  MoveC 1160 to (436.44, -29.66, -5) mm, rotated rx -180 ry 0 rz 5 deg; joints [27.358, -51.401, 157.25, 33.23, -102.458, 8.804] to (420.46, -17.39, -5) mm, rotated rx -180 ry 0 rz 0 deg; joints [25.818, -51.435, 156.847, 26.539, -102.977, 7.092]
  MoveL 1161 to (395.06, -17.39, -5) mm, rotated rx -180 ry 0 rz 0 deg; joints [25.049, -51.607, 155.297, 25.593, -101.516, 6.141]
  MoveL 1162 to (318.86, -17.39, -5) mm, rotated rx -180 ry 0 rz 0 deg; joints [22.982, -51.648, 150.513, 23.174, -97.289, 3.75]
  MoveC 1163 to (306.16, -30.09, -5) mm, rotated rx 180 ry 0 rz 0 deg; joints [21.924, -51.604, 150.031, 22.088, -96.946, 3.432] to (293.46, -17.39, -5) mm, rotated rx -180 ry 0 rz 0 deg; joints [22.363, -51.526, 148.876, 22.483, -95.926, 3.077]
  MoveL 1164 to (191.86, -17.39, -5) mm, rotated rx -180 ry 0 rz 0 deg; joints [20.176, -50.499, 142.119, 20.171, -90.651, 0.831]
  MoveC 1165 to (179.16, -30.09, -5) mm, rotated rx -180 ry 0 rz 0 deg; joints [19.26, -50.373, 141.56, 19.254, -90.251, 0.664] to (166.46, -17.39, -5) mm, rotated rx -180 ry 0 rz 0 deg; joints [19.692, -50.127, 140.379, 19.686, -89.368, 0.357]
  MoveL 1166 to (90.26, -17.39, -5) mm, rotated rx 180 ry 0 rz 0 deg; joints [18.365, -48.779, 135.036, 18.415, -85.578, -0.909]
  MoveL 1167 to (64.86, -17.39, -5) mm, rotated rx -180 ry 0 rz 0 deg; joints [17.96, -48.259, 133.212, 18.045, -84.33, -1.289]
  MoveC 1168 to (61.14, -26.37, -5) mm, rotated rx -180 ry 0 rz 0 deg; joints [17.47, -48.234, 133.149, 17.554, -84.28, -1.26] to (52.16, -30.09, -5) mm, rotated rx 180 ry 0 rz 0 deg; joints [17.156, -48.064, 132.58, 17.251, -83.891, -1.352]
  MoveL 1169 to (52.16, -30.09, -5) mm, rotated rx 180 ry 0 rz 0 deg; joints [17.156, -48.064, 132.58, 17.251, -83.891, -1.352]
  MoveC 1170 to (43.18, -26.37, -5) mm, rotated rx 180 ry 0 rz 0 deg; joints [17.202, -47.846, 131.842, 17.314, -83.396, -1.512] to (39.46, -17.39, -5) mm, rotated rx -180 ry 0 rz 0 deg; joints [17.572, -47.707, 131.366, 17.699, -83.087, -1.652]
  MoveL 1171 to (14.06, -17.39, -5) mm, rotated rx 180 ry 0 rz 0 deg; joints [17.2, -47.124, 129.497, 17.375, -81.847, -1.999]
  MoveC 1172 to (13.61, -17.2, -5) mm, rotated rx -180 ry 0 rz 0 deg; joints [17.202, -47.112, 129.46, 17.378, -81.823, -2.007] to (13.42, -16.75, -5) mm, rotated rx -180 ry 0 rz 0 deg; joints [17.22, -47.105, 129.436, 17.397, -81.807, -2.015]
  MoveL 1173 to (13.42, -16.12, -5) mm, rotated rx 180 ry 0 rz 0 deg; joints [17.25, -47.101, 129.421, 17.428, -81.799, -2.022]
  MoveC 1174 to (13.42, -15.67, -4.81) mm, rotated rx 180 ry 0 rz 0 deg; joints [17.271, -47.111, 129.414, 17.449, -81.782, -2.03] to (13.42, -15.48, -4.37) mm, rotated rx -180 ry 0 rz 0 deg; joints [17.279, -47.143, 129.416, 17.459, -81.755, -2.04]
  Set speed (500.0 mm/s)
  MoveL 1175 to (13.42, -15.48, 5) mm, rotated rx 180 ry 0 rz 0 deg; joints [17.275, -47.829, 129.55, 17.48, -81.228, -2.207]
  MoveL 1176 to (12.15, -16.75, 5) mm, rotated rx -180 ry 0 rz 0 deg; joints [17.198, -47.807, 129.485, 17.404, -81.184, -2.209]
  Set speed (25.4 mm/s)
  MoveL 1177 to (12.15, -16.75, 1) mm, rotated rx 180 ry 0 rz 0 deg; joints [17.2, -47.515, 129.429, 17.395, -81.409, -2.138]
  MoveL 1178 to (12.15, -16.75, -7.72) mm, rotated rx -180 ry 0 rz 0 deg; joints [17.203, -46.876, 129.301, 17.376, -81.897, -1.984]
  MoveC 1179 to (12.34, -16.75, -8.16) mm, rotated rx 180 ry 0 rz 0 deg; joints [17.206, -46.847, 129.308, 17.378, -81.931, -1.974] to (12.79, -16.75, -8.35) mm, rotated rx -180 ry 0 rz 0 deg; joints [17.213, -46.844, 129.338, 17.383, -81.963, -1.964]
  Set speed (50.8 mm/s)
  MoveL 1180 to (13.42, -16.75, -8.35) mm, rotated rx 180 ry 0 rz 0 deg; joints [17.222, -46.859, 129.385, 17.391, -81.994, -1.956]
  MoveC 1181 to (13.87, -16.94, -8.35) mm, rotated rx -180 ry 0 rz 0 deg; joints [17.22, -46.871, 129.423, 17.387, -82.019, -1.948] to (14.06, -17.39, -8.35) mm, rotated rx -180 ry 0 rz 0 deg; joints [17.202, -46.878, 129.447, 17.368, -82.034, -1.941]
  MoveL 1182 to (14.06, -169.79, -8.35) mm, rotated rx 180 ry 0 rz 0 deg; joints [9.897, -47.619, 132.176, 9.952, -83.768, -0.667]
  MoveL 1183 to (471.26, -169.79, -8.35) mm, rotated rx 180 ry 0 rz 30 deg; joints [26.906, -51.035, 156.836, 57.701, -97.685, 13.109]
  MoveL 1184 to (471.26, -17.39, -8.35) mm, rotated rx 180 ry 0 rz 30 deg; joints [35.788, -51.568, 151.463, 65.967, -93.163, 8.832]
  MoveL 1185 to (445.86, -17.39, -8.35) mm, rotated rx -180 ry 0 rz 30 deg; joints [34.843, -51.495, 150.022, 64.967, -92.733, 7.523]
  MoveC 1186 to (436.44, -29.66, -8.35) mm, rotated rx -180 ry 0 rz 5 deg; joints [27.361, -50.987, 157.17, 33.274, -102.738, 8.992] to (420.46, -17.39, -8.35) mm, rotated rx -180 ry 0 rz 0 deg; joints [25.82, -51.025, 156.767, 26.576, -103.273, 7.245]
  MoveL 1187 to (395.06, -17.39, -8.35) mm, rotated rx -180 ry 0 rz 0 deg; joints [25.052, -51.212, 155.221, 25.624, -101.804, 6.282]
  MoveL 1188 to (318.86, -17.39, -8.35) mm, rotated rx -180 ry 0 rz 0 deg; joints [22.985, -51.293, 150.445, 23.19, -97.552, 3.864]
  MoveC 1189 to (306.16, -30.09, -8.35) mm, rotated rx -180 ry 0 rz 0 deg; joints [21.926, -51.253, 149.963, 22.103, -97.208, 3.539] to (293.46, -17.39, -8.35) mm, rotated rx -180 ry 0 rz 0 deg; joints [22.366, -51.184, 148.809, 22.497, -96.181, 3.183]
  MoveL 1190 to (191.86, -17.39, -8.35) mm, rotated rx -180 ry 0 rz 0 deg; joints [20.178, -50.199, 142.06, 20.174, -90.878, 0.914]
  MoveC 1191 to (179.16, -30.09, -8.35) mm, rotated rx -180 ry 0 rz 0 deg; joints [19.262, -50.075, 141.501, 19.256, -90.477, 0.743] to (166.46, -17.39, -8.35) mm, rotated rx -180 ry 0 rz 0 deg; joints [19.693, -49.836, 140.322, 19.687, -89.588, 0.436]
  MoveL 1192 to (90.26, -17.39, -8.35) mm, rotated rx -180 ry 0 rz 0 deg; joints [18.366, -48.512, 134.982, 18.412, -85.781, -0.842]
  MoveL 1193 to (64.86, -17.39, -8.35) mm, rotated rx -180 ry 0 rz 0 deg; joints [17.961, -47.999, 133.16, 18.04, -84.527, -1.225]
  MoveC 1194 to (61.14, -26.37, -8.35) mm, rotated rx 180 ry 0 rz 0 deg; joints [17.472, -47.975, 133.097, 17.549, -84.478, -1.197] to (52.16, -30.09, -8.35) mm, rotated rx 180 ry 0 rz 0 deg; joints [17.158, -47.807, 132.528, 17.246, -84.088, -1.291]
  MoveL 1195 to (52.16, -30.09, -8.35) mm, rotated rx 180 ry 0 rz 0 deg; joints [17.158, -47.807, 132.528, 17.246, -84.088, -1.291]
  MoveC 1196 to (43.18, -26.37, -8.35) mm, rotated rx 180 ry 0 rz 0 deg; joints [17.203, -47.591, 131.79, 17.309, -83.59, -1.451] to (39.46, -17.39, -8.35) mm, rotated rx 180 ry 0 rz 0 deg; joints [17.574, -47.454, 131.315, 17.693, -83.279, -1.591]
  MoveL 1197 to (14.06, -17.39, -8.35) mm, rotated rx -180 ry 0 rz 0 deg; joints [17.202, -46.878, 129.447, 17.368, -82.034, -1.941]
  MoveC 1198 to (13.61, -17.2, -8.35) mm, rotated rx -180 ry 0 rz 0 deg; joints [17.204, -46.866, 129.409, 17.372, -82.009, -1.949] to (13.42, -16.75, -8.35) mm, rotated rx -180 ry 0 rz 0 deg; joints [17.222, -46.859, 129.385, 17.391, -81.994, -1.956]
  MoveL 1199 to (13.42, -16.12, -8.35) mm, rotated rx -180 ry 0 rz 0 deg; joints [17.251, -46.855, 129.371, 17.421, -81.986, -1.963]
  MoveC 1200 to (13.42, -15.67, -8.16) mm, rotated rx -180 ry 0 rz 0 deg; joints [17.272, -46.866, 129.363, 17.442, -81.969, -1.971] to (13.42, -15.48, -7.72) mm, rotated rx 180 ry 0 rz 0 deg; joints [17.28, -46.897, 129.366, 17.452, -81.941, -1.981]
  Set speed (500.0 mm/s)
  MoveL 1201 to (13.42, -15.48, 6) mm, rotated rx 180 ry 0 rz 0 deg; joints [17.274, -47.903, 129.564, 17.482, -81.171, -2.225]
  MoveL 1202 to (-18.41, -15.48, 6) mm, rotated rx -180 ry 0 rz 0 deg; joints [16.828, -47.103, 127.185, 17.109, -79.642, -2.632]
  Set speed (25.4 mm/s)
  MoveL 1203 to (-18.41, -15.48, -4.36) mm, rotated rx 180 ry 0 rz 0 deg; joints [16.832, -46.367, 127.04, 17.083, -80.207, -2.457]
  MoveC 1204 to (-18.41, -15.67, -4.81) mm, rotated rx -180 ry 0 rz 0 deg; joints [16.824, -46.337, 127.038, 17.073, -80.234, -2.447] to (-18.41, -16.12, -5) mm, rotated rx 180 ry 0 rz 0 deg; joints [16.804, -46.327, 127.045, 17.051, -80.249, -2.439]
  Set speed (50.8 mm/s)
  MoveL 1205 to (-18.41, -16.75, -5) mm, rotated rx 180 ry 0 rz 0 deg; joints [16.775, -46.331, 127.06, 17.022, -80.258, -2.431]
  MoveC 1206 to (-18.6, -17.2, -5) mm, rotated rx 180 ry 0 rz 0 deg; joints [16.752, -46.33, 127.056, 16.999, -80.254, -2.428] to (-19.04, -17.39, -5) mm, rotated rx -180 ry 0 rz 0 deg; joints [16.738, -46.32, 127.026, 16.985, -80.235, -2.432]
  MoveL 1207 to (-39.46, -17.39, -5) mm, rotated rx -180 ry 0 rz 0 deg; joints [16.465, -45.799, 125.482, 16.762, -79.242, -2.689]
  MoveC 1208 to (-52.16, -30.09, -5) mm, rotated rx -180 ry 0 rz 0 deg; joints [15.736, -45.554, 124.79, 16.045, -78.775, -2.687] to (-64.86, -17.39, -5) mm, rotated rx -180 ry 0 rz 0 deg; joints [16.136, -45.126, 123.537, 16.501, -78.005, -2.999]
  MoveL 1209 to (-90.26, -17.39, -5) mm, rotated rx 180 ry 0 rz 0 deg; joints [15.821, -44.425, 121.565, 16.258, -76.767, -3.301]
  MoveL 1210 to (-166.46, -17.39, -5) mm, rotated rx -180 ry 0 rz 0 deg; joints [14.942, -42.16, 115.477, 15.633, -73.03, -4.165]
  MoveC 1211 to (-179.16, -30.09, -5) mm, rotated rx -180 ry 0 rz 0 deg; joints [14.289, -41.857, 114.706, 14.99, -72.527, -4.103] to (-191.86, -17.39, -5) mm, rotated rx -180 ry 0 rz 0 deg; joints [14.67, -41.351, 113.385, 15.458, -71.772, -4.444]
  MoveL 1212 to (-293.46, -17.39, -5) mm, rotated rx -180 ry 0 rz 0 deg; joints [13.673, -37.838, 104.651, 14.914, -66.642, -5.544]
  MoveC 1213 to (-306.16, -30.09, -5) mm, rotated rx 180 ry 0 rz 0 deg; joints [13.081, -37.473, 103.782, 14.328, -66.095, -5.435] to (-318.86, -17.39, -5) mm, rotated rx 180 ry 0 rz 0 deg; joints [13.444, -36.887, 102.363, 14.818, -65.326, -5.822]
  MoveL 1214 to (-395.06, -17.39, -5) mm, rotated rx -180 ry 0 rz 0 deg; joints [12.8, -33.84, 95.197, 14.628, -61.268, -6.682]
  MoveL 1215 to (-420.46, -17.39, -5) mm, rotated rx -180 ry 0 rz 0 deg; joints [12.599, -32.754, 92.693, 14.601, -59.871, -6.983]
  MoveC 1216 to (-433.16, -30.09, -5) mm, rotated rx -180 ry 0 rz 0 deg; joints [12.059, -32.314, 91.695, 14.061, -59.263, -6.837] to (-445.86, -17.39, -5) mm, rotated rx -180 ry 0 rz 0 deg; joints [12.404, -31.629, 90.122, 14.593, -58.447, -7.295]
  MoveL 1217 to (-471.26, -17.39, -5) mm, rotated rx -180 ry 0 rz 0 deg; joints [12.214, -30.463, 87.478, 14.606, -56.991, -7.62]
  MoveL 1218 to (-471.26, -169.79, -5) mm, rotated rx -180 ry 0 rz 0 deg; joints [6.956, -31.599, 90.168, 8.208, -57.959, -3.998]
  MoveL 1219 to (-14.06, -169.79, -5) mm, rotated rx -180 ry 0 rz 0 deg; joints [9.66, -47.226, 130.101, 9.748, -82.107, -0.931]
  MoveL 1220 to (-14.06, -17.39, -5) mm, rotated rx -180 ry 0 rz 0 deg; joints [16.806, -46.444, 127.401, 17.042, -80.478, -2.368]
  MoveL 1221 to (-19.04, -17.39, -5) mm, rotated rx -180 ry 0 rz 0 deg; joints [16.738, -46.32, 127.026, 16.985, -80.235, -2.432]
  MoveC 1222 to (-19.49, -17.2, -5) mm, rotated rx -180 ry 0 rz 0 deg; joints [16.74, -46.307, 126.988, 16.989, -80.211, -2.44] to (-19.68, -16.75, -5) mm, rotated rx 180 ry 0 rz 0 deg; joints [16.758, -46.299, 126.964, 17.008, -80.196, -2.447]
  MoveL 1223 to (-19.68, -16.12, -5) mm, rotated rx 180 ry 0 rz 0 deg; joints [16.787, -46.295, 126.95, 17.037, -80.188, -2.455]
  MoveC 1224 to (-19.68, -15.67, -4.81) mm, rotated rx 180 ry 0 rz 0 deg; joints [16.807, -46.305, 126.942, 17.058, -80.172, -2.463] to (-19.68, -15.48, -4.37) mm, rotated rx -180 ry 0 rz 0 deg; joints [16.815, -46.336, 126.945, 17.068, -80.145, -2.473]
  Set speed (500.0 mm/s)
  MoveL 1225 to (-19.68, -15.48, 5) mm, rotated rx -180 ry 0 rz 0 deg; joints [16.811, -46.999, 127.076, 17.092, -79.636, -2.631]
  MoveL 1226 to (-18.41, -15.48, 5) mm, rotated rx 180 ry 0 rz 0 deg; joints [16.828, -47.032, 127.172, 17.106, -79.697, -2.615]
  Set speed (25.4 mm/s)
  MoveL 1227 to (-18.41, -15.48, 1) mm, rotated rx 180 ry 0 rz 0 deg; joints [16.83, -46.748, 127.116, 17.096, -79.916, -2.547]
  MoveL 1228 to (-18.41, -15.48, -7.71) mm, rotated rx 180 ry 0 rz 0 deg; joints [16.834, -46.129, 126.991, 17.075, -80.388, -2.401]
  MoveC 1229 to (-18.41, -15.67, -8.16) mm, rotated rx -180 ry 0 rz 0 deg; joints [16.826, -46.099, 126.989, 17.065, -80.414, -2.391] to (-18.41, -16.12, -8.35) mm, rotated rx -180 ry 0 rz 0 deg; joints [16.805, -46.089, 126.996, 17.043, -80.43, -2.383]
  Set speed (50.8 mm/s)
  MoveL 1230 to (-18.41, -16.75, -8.35) mm, rotated rx -180 ry 0 rz 0 deg; joints [16.777, -46.093, 127.011, 17.014, -80.438, -2.375]
  MoveC 1231 to (-18.6, -17.2, -8.35) mm, rotated rx -180 ry 0 rz 0 deg; joints [16.754, -46.091, 127.007, 16.991, -80.435, -2.373] to (-19.04, -17.39, -8.35) mm, rotated rx 180 ry 0 rz 0 deg; joints [16.739, -46.081, 126.977, 16.977, -80.416, -2.376]
  MoveL 1232 to (-39.46, -17.39, -8.35) mm, rotated rx -180 ry 0 rz 0 deg; joints [16.466, -45.566, 125.433, 16.753, -79.419, -2.635]
  MoveC 1233 to (-52.16, -30.09, -8.35) mm, rotated rx -180 ry 0 rz 0 deg; joints [15.737, -45.323, 124.742, 16.036, -78.951, -2.636] to (-64.86, -17.39, -8.35) mm, rotated rx -180 ry 0 rz 0 deg; joints [16.138, -44.898, 123.489, 16.491, -78.178, -2.947]
  MoveL 1234 to (-90.26, -17.39, -8.35) mm, rotated rx -180 ry 0 rz 0 deg; joints [15.822, -44.203, 121.518, 16.248, -76.935, -3.25]
  MoveL 1235 to (-166.46, -17.39, -8.35) mm, rotated rx 180 ry 0 rz 0 deg; joints [14.943, -41.952, 115.432, 15.621, -73.186, -4.12]
  MoveC 1236 to (-179.16, -30.09, -8.35) mm, rotated rx -180 ry 0 rz 0 deg; joints [14.29, -41.651, 114.66, 14.978, -72.683, -4.059] to (-191.86, -17.39, -8.35) mm, rotated rx -180 ry 0 rz 0 deg; joints [14.671, -41.148, 113.34, 15.445, -71.925, -4.4]
  MoveL 1237 to (-293.46, -17.39, -8.35) mm, rotated rx -180 ry 0 rz 0 deg; joints [13.674, -37.65, 104.607, 14.899, -66.781, -5.504]
  MoveC 1238 to (-306.16, -30.09, -8.35) mm, rotated rx -180 ry 0 rz 0 deg; joints [13.083, -37.286, 103.738, 14.313, -66.233, -5.397] to (-318.86, -17.39, -8.35) mm, rotated rx -180 ry 0 rz 0 deg; joints [13.445, -36.702, 102.319, 14.802, -65.462, -5.783]
  MoveL 1239 to (-395.06, -17.39, -8.35) mm, rotated rx 180 ry 0 rz 0 deg; joints [12.801, -33.665, 95.153, 14.611, -61.395, -6.644]
  MoveL 1240 to (-420.46, -17.39, -8.35) mm, rotated rx -180 ry 0 rz 0 deg; joints [12.6, -32.582, 92.649, 14.583, -59.995, -6.946]
  MoveC 1241 to (-433.16, -30.09, -8.35) mm, rotated rx -180 ry 0 rz 0 deg; joints [12.06, -32.143, 91.65, 14.044, -59.386, -6.802] to (-445.86, -17.39, -8.35) mm, rotated rx -180 ry 0 rz 0 deg; joints [12.405, -31.46, 90.078, 14.575, -58.568, -7.258]
  MoveL 1242 to (-471.26, -17.39, -8.35) mm, rotated rx -180 ry 0 rz 0 deg; joints [12.215, -30.296, 87.433, 14.588, -57.11, -7.583]
  MoveL 1243 to (-471.26, -169.79, -8.35) mm, rotated rx -180 ry 0 rz 0 deg; joints [6.957, -31.429, 90.123, 8.198, -58.082, -3.977]
  MoveL 1244 to (-14.06, -169.79, -8.35) mm, rotated rx 180 ry 0 rz 0 deg; joints [9.661, -46.978, 130.051, 9.745, -82.302, -0.898]
  MoveL 1245 to (-14.06, -17.39, -8.35) mm, rotated rx -180 ry 0 rz 0 deg; joints [16.807, -46.205, 127.352, 17.034, -80.659, -2.312]
  MoveL 1246 to (-19.04, -17.39, -8.35) mm, rotated rx 180 ry 0 rz 0 deg; joints [16.739, -46.081, 126.977, 16.977, -80.416, -2.376]
  MoveC 1247 to (-19.49, -17.2, -8.35) mm, rotated rx -180 ry 0 rz 0 deg; joints [16.741, -46.069, 126.939, 16.981, -80.391, -2.384] to (-19.68, -16.75, -8.35) mm, rotated rx -180 ry 0 rz 0 deg; joints [16.759, -46.061, 126.915, 16.999, -80.376, -2.392]
  MoveL 1248 to (-19.68, -16.12, -8.35) mm, rotated rx -180 ry 0 rz 0 deg; joints [16.788, -46.057, 126.901, 17.029, -80.368, -2.399]
  MoveC 1249 to (-19.68, -15.67, -8.16) mm, rotated rx -180 ry 0 rz 0 deg; joints [16.808, -46.067, 126.893, 17.05, -80.352, -2.407] to (-19.68, -15.48, -7.72) mm, rotated rx -180 ry 0 rz 0 deg; joints [16.816, -46.098, 126.896, 17.06, -80.326, -2.417]
  Set speed (500.0 mm/s)
  MoveL 1250 to (-19.68, -15.48, 6) mm, rotated rx -180 ry 0 rz 0 deg; joints [16.811, -47.07, 127.09, 17.095, -79.581, -2.648]
  MoveL 1251 to (-13.42, -196.52, 6) mm, rotated rx 180 ry 0 rz 0 deg; joints [8.369, -48.146, 130.629, 8.453, -81.694, -0.83]
  Set speed (25.4 mm/s)
  MoveL 1252 to (-13.42, -196.51, -4.36) mm, rotated rx -180 ry 0 rz 0 deg; joints [8.373, -47.375, 130.479, 8.444, -82.309, -0.738]
  MoveC 1253 to (-13.42, -196.7, -4.81) mm, rotated rx -180 ry 0 rz 0 deg; joints [8.364, -47.342, 130.474, 8.435, -82.336, -0.733] to (-13.42, -197.15, -5) mm, rotated rx 180 ry 0 rz 0 deg; joints [8.342, -47.329, 130.477, 8.412, -82.351, -0.728]
  Set speed (50.8 mm/s)
  MoveL 1254 to (-13.42, -197.78, -5) mm, rotated rx -180 ry 0 rz 0 deg; joints [8.311, -47.331, 130.484, 8.381, -82.355, -0.724]
  MoveC 1255 to (-13.61, -198.23, -5) mm, rotated rx -180 ry 0 rz 0 deg; joints [8.288, -47.328, 130.474, 8.358, -82.349, -0.722] to (-14.06, -198.42, -5) mm, rotated rx 180 ry 0 rz 0 deg; joints [8.276, -47.318, 130.442, 8.346, -82.327, -0.723]
  MoveL 1256 to (-39.46, -198.42, -5) mm, rotated rx 180 ry 0 rz 0 deg; joints [8.101, -46.702, 128.494, 8.197, -81.005, -0.894]
  MoveC 1257 to (-52.16, -211.12, -5) mm, rotated rx -180 ry 0 rz 0 deg; joints [7.417, -46.42, 127.644, 7.518, -80.428, -0.872] to (-64.86, -198.42, -5) mm, rotated rx -180 ry 0 rz 0 deg; joints [7.932, -46.056, 126.524, 8.058, -79.691, -1.058]
  MoveL 1258 to (-90.26, -198.42, -5) mm, rotated rx -180 ry 0 rz 0 deg; joints [7.771, -45.379, 124.529, 7.93, -78.381, -1.216]
  MoveL 1259 to (-166.46, -198.42, -5) mm, rotated rx -180 ry 0 rz 0 deg; joints [7.324, -43.178, 118.39, 7.598, -74.466, -1.662]
  MoveC 1260 to (-179.16, -211.12, -5) mm, rotated rx -180 ry 0 rz 0 deg; joints [6.712, -42.83, 117.47, 6.983, -73.878, -1.573] to (-191.86, -198.42, -5) mm, rotated rx -180 ry 0 rz 0 deg; joints [7.186, -42.389, 116.287, 7.505, -73.159, -1.804]
  MoveL 1261 to (-293.46, -198.42, -5) mm, rotated rx -180 ry 0 rz 0 deg; joints [6.683, -38.95, 107.539, 7.211, -67.872, -2.355]
  MoveC 1262 to (-306.16, -211.12, -5) mm, rotated rx -180 ry 0 rz 0 deg; joints [6.128, -38.535, 106.529, 6.642, -67.257, -2.212] to (-318.86, -198.42, -5) mm, rotated rx -180 ry 0 rz 0 deg; joints [6.567, -38.018, 105.256, 7.158, -66.527, -2.491]
  MoveL 1263 to (-395.06, -198.42, -5) mm, rotated rx -180 ry 0 rz 0 deg; joints [6.245, -35.036, 98.132, 7.045, -62.4, -2.909]
  MoveL 1264 to (-420.46, -198.42, -5) mm, rotated rx -180 ry 0 rz 0 deg; joints [6.144, -33.974, 95.651, 7.024, -60.986, -3.054]
  MoveC 1265 to (-433.16, -211.12, -5) mm, rotated rx 180 ry 0 rz 0 deg; joints [5.638, -33.482, 94.518, 6.487, -60.321, -2.864] to (-445.86, -198.42, -5) mm, rotated rx 180 ry 0 rz 0 deg; joints [6.047, -32.876, 93.11, 7.013, -59.549, -3.203]
  MoveL 1266 to (-471.26, -198.42, -5) mm, rotated rx -180 ry 0 rz 0 deg; joints [5.952, -31.738, 90.502, 7.012, -58.084, -3.357]
  MoveL 1267 to (-471.26, -350.82, -5) mm, rotated rx 180 ry 0 rz 0 deg; joints [0.562, -32.088, 91.393, 0.654, -58.436, -0.062]
  MoveL 1268 to (-14.06, -350.82, -5) mm, rotated rx -180 ry 0 rz 0 deg; joints [0.782, -47.534, 131.354, 0.784, -82.952, 0.188]
  MoveL 1269 to (-14.06, -198.42, -5) mm, rotated rx 180 ry 0 rz 0 deg; joints [8.276, -47.318, 130.442, 8.346, -82.327, -0.723]
  MoveC 1270 to (-13.87, -197.97, -5) mm, rotated rx 180 ry 0 rz 0 deg; joints [8.299, -47.321, 130.451, 8.369, -82.333, -0.725] to (-13.42, -197.78, -5) mm, rotated rx -180 ry 0 rz 0 deg; joints [8.311, -47.331, 130.484, 8.381, -82.355, -0.724]
  MoveL 1271 to (-12.79, -197.79, -5) mm, rotated rx 180 ry 0 rz 0 deg; joints [8.316, -47.346, 130.532, 8.385, -82.388, -0.719]
  MoveC 1272 to (-12.34, -197.79, -4.81) mm, rotated rx 180 ry 0 rz 0 deg; joints [8.319, -47.371, 130.569, 8.388, -82.401, -0.718] to (-12.15, -197.78, -4.37) mm, rotated rx -180 ry 0 rz 0 deg; joints [8.32, -47.409, 130.59, 8.39, -82.384, -0.72]
  Set speed (500.0 mm/s)
  MoveL 1273 to (-12.15, -197.79, 5) mm, rotated rx -180 ry 0 rz 0 deg; joints [8.317, -48.107, 130.726, 8.398, -81.828, -0.803]
  MoveL 1274 to (-13.42, -196.51, 5) mm, rotated rx 180 ry 0 rz 0 deg; joints [8.37, -48.072, 130.615, 8.452, -81.754, -0.821]
  Set speed (25.4 mm/s)
  MoveL 1275 to (-13.42, -196.51, 1) mm, rotated rx -180 ry 0 rz 0 deg; joints [8.371, -47.774, 130.558, 8.449, -81.992, -0.785]
  MoveL 1276 to (-13.42, -196.51, -7.71) mm, rotated rx -180 ry 0 rz 0 deg; joints [8.374, -47.125, 130.428, 8.441, -82.505, -0.709]
  MoveC 1277 to (-13.42, -196.7, -8.16) mm, rotated rx -180 ry 0 rz 0 deg; joints [8.365, -47.092, 130.424, 8.432, -82.533, -0.703] to (-13.42, -197.15, -8.35) mm, rotated rx -180 ry 0 rz 0 deg; joints [8.343, -47.08, 130.426, 8.41, -82.547, -0.699]
  Set speed (50.8 mm/s)
  MoveL 1278 to (-13.42, -197.78, -8.35) mm, rotated rx -180 ry 0 rz 0 deg; joints [8.312, -47.082, 130.433, 8.379, -82.552, -0.694]
  MoveC 1279 to (-13.61, -198.23, -8.35) mm, rotated rx 180 ry 0 rz 0 deg; joints [8.289, -47.079, 130.424, 8.355, -82.545, -0.693] to (-14.06, -198.42, -8.35) mm, rotated rx -180 ry 0 rz 0 deg; joints [8.277, -47.069, 130.391, 8.343, -82.523, -0.695]
  MoveL 1280 to (-39.46, -198.42, -8.35) mm, rotated rx -180 ry 0 rz 0 deg; joints [8.102, -46.459, 128.444, 8.194, -81.196, -0.866]
  MoveC 1281 to (-52.16, -211.12, -8.35) mm, rotated rx 180 ry 0 rz 0 deg; joints [7.418, -46.18, 127.595, 7.515, -80.617, -0.846] to (-64.86, -198.42, -8.35) mm, rotated rx -180 ry 0 rz 0 deg; joints [7.934, -45.819, 126.475, 8.055, -79.876, -1.031]
  MoveL 1282 to (-90.26, -198.42, -8.35) mm, rotated rx -180 ry 0 rz 0 deg; joints [7.772, -45.149, 124.481, 7.925, -78.562, -1.19]
  MoveL 1283 to (-166.46, -198.42, -8.35) mm, rotated rx -180 ry 0 rz 0 deg; joints [7.325, -42.964, 118.344, 7.593, -74.633, -1.639]
  MoveC 1284 to (-179.16, -211.12, -8.35) mm, rotated rx 180 ry 0 rz 0 deg; joints [6.713, -42.618, 117.424, 6.978, -74.044, -1.552] to (-191.86, -198.42, -8.35) mm, rotated rx 180 ry 0 rz 0 deg; joints [7.187, -42.179, 116.241, 7.499, -73.321, -1.782]
  MoveL 1285 to (-293.46, -198.42, -8.35) mm, rotated rx 180 ry 0 rz 0 deg; joints [6.683, -38.757, 107.494, 7.205, -68.019, -2.335]
  MoveC 1286 to (-306.16, -211.12, -8.35) mm, rotated rx -180 ry 0 rz 0 deg; joints [6.129, -38.344, 106.485, 6.636, -67.403, -2.194] to (-318.86, -198.42, -8.35) mm, rotated rx -180 ry 0 rz 0 deg; joints [6.568, -37.829, 105.212, 7.151, -66.67, -2.472]
  MoveL 1287 to (-395.06, -198.42, -8.35) mm, rotated rx -180 ry 0 rz 0 deg; joints [6.246, -34.857, 98.088, 7.037, -62.534, -2.891]
  MoveL 1288 to (-420.46, -198.42, -8.35) mm, rotated rx -180 ry 0 rz 0 deg; joints [6.145, -33.798, 95.607, 7.016, -61.117, -3.036]
  MoveC 1289 to (-433.16, -211.12, -8.35) mm, rotated rx -180 ry 0 rz 0 deg; joints [5.639, -33.307, 94.474, 6.48, -60.451, -2.848] to (-445.86, -198.42, -8.35) mm, rotated rx -180 ry 0 rz 0 deg; joints [6.047, -32.703, 93.066, 7.005, -59.676, -3.185]
  MoveL 1290 to (-471.26, -198.42, -8.35) mm, rotated rx -180 ry 0 rz 0 deg; joints [5.953, -31.568, 90.458, 7.003, -58.209, -3.34]
  MoveL 1291 to (-471.26, -350.82, -8.35) mm, rotated rx 180 ry 0 rz 0 deg; joints [0.562, -31.917, 91.348, 0.654, -58.563, -0.06]
  MoveL 1292 to (-14.06, -350.82, -8.35) mm, rotated rx -180 ry 0 rz 0 deg; joints [0.783, -47.281, 131.303, 0.784, -83.153, 0.191]
  MoveL 1293 to (-14.06, -198.42, -8.35) mm, rotated rx -180 ry 0 rz 0 deg; joints [8.277, -47.069, 130.391, 8.343, -82.523, -0.695]
  MoveC 1294 to (-13.87, -197.97, -8.35) mm, rotated rx -180 ry 0 rz 0 deg; joints [8.3, -47.072, 130.401, 8.367, -82.53, -0.696] to (-13.42, -197.78, -8.35) mm, rotated rx -180 ry 0 rz 0 deg; joints [8.312, -47.082, 130.433, 8.379, -82.552, -0.694]
  MoveL 1295 to (-12.79, -197.78, -8.35) mm, rotated rx 180 ry 0 rz 0 deg; joints [8.317, -47.096, 130.481, 8.382, -82.585, -0.69]
  MoveC 1296 to (-12.34, -197.78, -8.16) mm, rotated rx -180 ry 0 rz 0 deg; joints [8.32, -47.121, 130.518, 8.385, -82.598, -0.689] to (-12.15, -197.78, -7.72) mm, rotated rx -180 ry 0 rz 0 deg; joints [8.321, -47.159, 130.539, 8.387, -82.581, -0.691]
  Set speed (500.0 mm/s)
  MoveL 1297 to (-12.15, -197.79, 6) mm, rotated rx -180 ry 0 rz 0 deg; joints [8.317, -48.181, 130.74, 8.399, -81.769, -0.812]
  MoveL 1298 to (12.15, -197.78, 6) mm, rotated rx -180 ry 0 rz 0 deg; joints [8.493, -48.76, 132.585, 8.551, -83.024, -0.644]
  Set speed (25.4 mm/s)
  MoveL 1299 to (12.15, -197.78, -4.36) mm, rotated rx -180 ry 0 rz 0 deg; joints [8.496, -47.967, 132.432, 8.544, -83.656, -0.549]
  MoveC 1300 to (12.34, -197.78, -4.81) mm, rotated rx -180 ry 0 rz 0 deg; joints [8.498, -47.937, 132.439, 8.545, -83.693, -0.543] to (12.79, -197.79, -5) mm, rotated rx 180 ry 0 rz 0 deg; joints [8.501, -47.932, 132.47, 8.548, -83.728, -0.538]
  Set speed (50.8 mm/s)
  MoveL 1301 to (13.42, -197.79, -5) mm, rotated rx 180 ry 0 rz 0 deg; joints [8.506, -47.946, 132.518, 8.552, -83.762, -0.534]
  MoveC 1302 to (13.87, -197.97, -5) mm, rotated rx -180 ry 0 rz 0 deg; joints [8.5, -47.957, 132.554, 8.546, -83.787, -0.529] to (14.06, -198.42, -5) mm, rotated rx 180 ry 0 rz 0 deg; joints [8.479, -47.962, 132.573, 8.524, -83.8, -0.525]
  MoveL 1303 to (14.06, -350.82, -5) mm, rotated rx -180 ry 0 rz 0 deg; joints [0.801, -48.164, 133.496, 0.801, -84.463, 0.207]
  MoveL 1304 to (471.26, -350.82, -5) mm, rotated rx 180 ry 0 rz -60 deg; joints [-17.821, -51.324, 151.408, -77.973, -91.92, -8.972]
  MoveL 1305 to (471.26, -198.42, -5) mm, rotated rx -180 ry 0 rz -60 deg; joints [-7.949, -51.323, 153.756, -68.382, -94.441, -10.657]
  MoveL 1306 to (445.86, -198.42, -5) mm, rotated rx 180 ry 0 rz -60 deg; joints [-7.718, -51.355, 152.031, -68.036, -93.831, -9.004]
  MoveC 1307 to (433.16, -211.12, -5) mm, rotated rx -180 ry 0 rz -60 deg; joints [-8.422, -51.332, 151.038, -68.675, -93.358, -8.147] to (420.46, -198.42, -5) mm, rotated rx -180 ry 0 rz -60 deg; joints [-7.5, -51.304, 150.288, -67.724, -93.229, -7.42]
  MoveL 1308 to (395.06, -198.42, -5) mm, rotated rx -180 ry 0 rz -30 deg; joints [0.228, -50.982, 157.395, -30.724, -103.586, -7.63]
  MoveL 1309 to (318.86, -198.42, -5) mm, rotated rx -180 ry 0 rz 0 deg; joints [11.543, -51.473, 154.194, 11.781, -101.591, 2.85]
  MoveC 1310 to (306.16, -211.12, -5) mm, rotated rx -180 ry 0 rz 0 deg; joints [10.534, -51.491, 153.507, 10.725, -100.942, 2.493] to (293.46, -198.42, -5) mm, rotated rx -180 ry 0 rz 0 deg; joints [11.207, -51.519, 152.489, 11.372, -99.89, 2.423]
  MoveL 1311 to (191.86, -198.42, -5) mm, rotated rx -180 ry 0 rz 0 deg; joints [10.035, -50.954, 145.495, 10.05, -93.602, 1.064]
  MoveC 1312 to (179.16, -211.12, -5) mm, rotated rx 180 ry 0 rz 0 deg; joints [9.17, -50.83, 144.75, 9.178, -93.001, 0.897] to (166.46, -198.42, -5) mm, rotated rx 180 ry 0 rz 0 deg; joints [9.779, -50.661, 143.704, 9.78, -92.129, 0.789]
  MoveL 1313 to (90.26, -198.42, -5) mm, rotated rx 180 ry 0 rz 0 deg; joints [9.083, -49.494, 138.223, 9.084, -87.875, 0.072]
  MoveL 1314 to (64.86, -198.42, -5) mm, rotated rx -180 ry 0 rz 0 deg; joints [8.873, -49.02, 136.359, 8.884, -86.501, -0.139]
  MoveC 1315 to (61.14, -207.4, -5) mm, rotated rx -180 ry 0 rz 0 deg; joints [8.377, -48.969, 136.184, 8.389, -86.375, -0.134] to (52.16, -211.12, -5) mm, rotated rx 180 ry 0 rz 0 deg; joints [8.118, -48.8, 135.558, 8.133, -85.921, -0.186]
  MoveL 1316 to (52.16, -211.12, -5) mm, rotated rx 180 ry 0 rz 0 deg; joints [8.118, -48.8, 135.558, 8.133, -85.921, -0.186]
  MoveC 1317 to (43.18, -207.4, -5) mm, rotated rx 180 ry 0 rz 0 deg; joints [8.242, -48.609, 134.851, 8.264, -85.412, -0.267] to (39.46, -198.42, -5) mm, rotated rx -180 ry 0 rz 0 deg; joints [8.671, -48.509, 134.476, 8.698, -85.143, -0.337]
  MoveL 1318 to (14.06, -198.42, -5) mm, rotated rx -180 ry 0 rz 0 deg; joints [8.479, -47.962, 132.573, 8.524, -83.8, -0.525]
  MoveC 1319 to (13.61, -198.23, -5) mm, rotated rx -180 ry 0 rz 0 deg; joints [8.485, -47.952, 132.537, 8.531, -83.775, -0.53] to (13.42, -197.79, -5) mm, rotated rx 180 ry 0 rz 0 deg; joints [8.506, -47.946, 132.518, 8.552, -83.762, -0.534]
  MoveL 1320 to (13.42, -197.15, -5) mm, rotated rx 180 ry 0 rz 0 deg; joints [8.538, -47.945, 132.511, 8.584, -83.757, -0.538]
  MoveC 1321 to (13.42, -196.7, -4.81) mm, rotated rx 180 ry 0 rz 0 deg; joints [8.56, -47.958, 132.509, 8.606, -83.742, -0.542] to (13.42, -196.52, -4.37) mm, rotated rx -180 ry 0 rz 0 deg; joints [8.569, -47.992, 132.513, 8.616, -83.714, -0.547]
  Set speed (500.0 mm/s)
  MoveL 1322 to (13.42, -196.51, 5) mm, rotated rx -180 ry 0 rz 0 deg; joints [8.566, -48.709, 132.653, 8.623, -83.142, -0.634]
  MoveL 1323 to (12.15, -197.79, 5) mm, rotated rx 180 ry 0 rz 0 deg; joints [8.493, -48.684, 132.571, 8.551, -83.085, -0.635]
  Set speed (25.4 mm/s)
  MoveL 1324 to (12.15, -197.78, 1) mm, rotated rx -180 ry 0 rz 0 deg; joints [8.494, -48.378, 132.513, 8.548, -83.33, -0.598]
  MoveL 1325 to (12.15, -197.78, -7.72) mm, rotated rx -180 ry 0 rz 0 deg; joints [8.498, -47.71, 132.38, 8.542, -83.859, -0.518]
  MoveC 1326 to (12.34, -197.79, -8.16) mm, rotated rx -180 ry 0 rz 0 deg; joints [8.499, -47.68, 132.387, 8.543, -83.896, -0.513] to (12.79, -197.79, -8.35) mm, rotated rx 180 ry 0 rz 0 deg; joints [8.502, -47.675, 132.418, 8.546, -83.931, -0.508]
  Set speed (50.8 mm/s)
  MoveL 1327 to (13.42, -197.79, -8.35) mm, rotated rx -180 ry 0 rz 0 deg; joints [8.507, -47.689, 132.466, 8.55, -83.965, -0.503]
  MoveC 1328 to (13.87, -197.97, -8.35) mm, rotated rx 180 ry 0 rz 0 deg; joints [8.501, -47.7, 132.502, 8.543, -83.99, -0.499] to (14.06, -198.42, -8.35) mm, rotated rx -180 ry 0 rz 0 deg; joints [8.48, -47.705, 132.521, 8.522, -84.003, -0.495]
  MoveL 1329 to (14.06, -350.82, -8.35) mm, rotated rx -180 ry 0 rz 0 deg; joints [0.802, -47.903, 133.444, 0.801, -84.671, 0.21]
  MoveL 1330 to (471.26, -350.82, -8.35) mm, rotated rx 180 ry 0 rz -60 deg; joints [-17.821, -50.962, 151.338, -77.983, -91.981, -9.257]
  MoveL 1331 to (471.26, -198.42, -8.35) mm, rotated rx 180 ry 0 rz -60 deg; joints [-7.948, -50.942, 153.682, -68.404, -94.554, -10.943]
  MoveL 1332 to (445.86, -198.42, -8.35) mm, rotated rx 180 ry 0 rz -60 deg; joints [-7.717, -50.988, 151.959, -68.054, -93.942, -9.278]
  MoveC 1333 to (433.16, -211.12, -8.35) mm, rotated rx -180 ry 0 rz -60 deg; joints [-8.421, -50.973, 150.968, -68.691, -93.463, -8.416] to (420.46, -198.42, -8.35) mm, rotated rx -180 ry 0 rz -60 deg; joints [-7.499, -50.951, 150.219, -67.738, -93.336, -7.683]
  MoveL 1334 to (395.06, -198.42, -8.35) mm, rotated rx -180 ry 0 rz -30 deg; joints [0.23, -50.566, 157.314, -30.764, -103.874, -7.806]
  MoveL 1335 to (318.86, -198.42, -8.35) mm, rotated rx -180 ry 0 rz 0 deg; joints [11.545, -51.088, 154.12, 11.796, -101.895, 2.915]
  MoveC 1336 to (306.16, -211.12, -8.35) mm, rotated rx 180 ry 0 rz 0 deg; joints [10.535, -51.112, 153.433, 10.738, -101.242, 2.551] to (293.46, -198.42, -8.35) mm, rotated rx -180 ry 0 rz 0 deg; joints [11.208, -51.149, 152.418, 11.385, -100.182, 2.483]
  MoveL 1337 to (191.86, -198.42, -8.35) mm, rotated rx -180 ry 0 rz 0 deg; joints [10.036, -50.634, 145.433, 10.054, -93.855, 1.109]
  MoveC 1338 to (179.16, -211.12, -8.35) mm, rotated rx -180 ry 0 rz 0 deg; joints [9.172, -50.515, 144.689, 9.182, -93.251, 0.938] to (166.46, -198.42, -8.35) mm, rotated rx 180 ry 0 rz 0 deg; joints [9.78, -50.352, 143.643, 9.784, -92.374, 0.831]
  MoveL 1339 to (90.26, -198.42, -8.35) mm, rotated rx 180 ry 0 rz 0 deg; joints [9.084, -49.213, 138.167, 9.084, -88.098, 0.107]
  MoveL 1340 to (64.86, -198.42, -8.35) mm, rotated rx -180 ry 0 rz 0 deg; joints [8.874, -48.747, 136.304, 8.883, -86.717, -0.105]
  MoveC 1341 to (61.14, -207.4, -8.35) mm, rotated rx -180 ry 0 rz 0 deg; joints [8.378, -48.697, 136.129, 8.388, -86.59, -0.102] to (52.16, -211.12, -8.35) mm, rotated rx -180 ry 0 rz 0 deg; joints [8.119, -48.531, 135.504, 8.132, -86.134, -0.156]
  MoveL 1342 to (52.16, -211.12, -8.35) mm, rotated rx -180 ry 0 rz 0 deg; joints [8.119, -48.531, 135.504, 8.132, -86.134, -0.156]
  MoveC 1343 to (43.18, -207.4, -8.35) mm, rotated rx -180 ry 0 rz 0 deg; joints [8.243, -48.342, 134.798, 8.263, -85.623, -0.237] to (39.46, -198.42, -8.35) mm, rotated rx -180 ry 0 rz 0 deg; joints [8.673, -48.244, 134.423, 8.696, -85.353, -0.305]
  MoveL 1344 to (14.06, -198.42, -8.35) mm, rotated rx -180 ry 0 rz 0 deg; joints [8.48, -47.705, 132.521, 8.522, -84.003, -0.495]
  MoveC 1345 to (13.61, -198.23, -8.35) mm, rotated rx 180 ry 0 rz 0 deg; joints [8.486, -47.695, 132.485, 8.529, -83.978, -0.499] to (13.42, -197.79, -8.35) mm, rotated rx -180 ry 0 rz 0 deg; joints [8.507, -47.689, 132.466, 8.55, -83.965, -0.503]
  MoveL 1346 to (13.42, -197.15, -8.35) mm, rotated rx -180 ry 0 rz 0 deg; joints [8.539, -47.688, 132.459, 8.582, -83.96, -0.507]
  MoveC 1347 to (13.42, -196.7, -8.16) mm, rotated rx -180 ry 0 rz 0 deg; joints [8.561, -47.701, 132.457, 8.604, -83.945, -0.511] to (13.42, -196.52, -7.72) mm, rotated rx 180 ry 0 rz 0 deg; joints [8.57, -47.735, 132.462, 8.614, -83.916, -0.516]
  Set speed (500.0 mm/s)
  MoveL 1348 to (13.42, -196.52, 6) mm, rotated rx 180 ry 0 rz 0 deg; joints [8.565, -48.786, 132.667, 8.623, -83.08, -0.644]
  MoveL 1349 to (12.15, -384.12, 6) mm, rotated rx -180 ry 0 rz 0 deg; joints [-0.891, -48.964, 133.513, -0.901, -83.68, 0.358]
  Set speed (25.4 mm/s)
  MoveL 1350 to (12.15, -384.12, -4.37) mm, rotated rx -180 ry 0 rz 0 deg; joints [-0.889, -48.159, 133.357, -0.897, -84.329, 0.347]
  MoveC 1351 to (12.34, -384.12, -4.81) mm, rotated rx -180 ry 0 rz 0 deg; joints [-0.889, -48.128, 133.364, -0.897, -84.367, 0.347] to (12.79, -384.12, -5) mm, rotated rx -180 ry 0 rz 0 deg; joints [-0.889, -48.124, 133.395, -0.897, -84.403, 0.346]
  Set speed (50.8 mm/s)
  MoveL 1352 to (13.42, -384.12, -5) mm, rotated rx 180 ry 0 rz 0 deg; joints [-0.89, -48.137, 133.444, -0.898, -84.437, 0.346]
  MoveC 1353 to (13.87, -384.31, -5) mm, rotated rx 180 ry 0 rz 0 deg; joints [-0.899, -48.147, 133.477, -0.908, -84.461, 0.346] to (14.06, -384.76, -5) mm, rotated rx -180 ry 0 rz 0 deg; joints [-0.922, -48.151, 133.491, -0.931, -84.471, 0.348]
  MoveL 1354 to (14.06, -537.16, -5) mm, rotated rx -180 ry 0 rz 0 deg; joints [-8.598, -47.831, 132.519, -8.65, -83.879, 1.07]
  MoveL 1355 to (471.26, -537.16, -5) mm, rotated rx -180 ry 0 rz -30 deg; joints [-25.102, -50.905, 157.482, -56.092, -98.794, -13.027]
  MoveL 1356 to (471.26, -384.76, -5) mm, rotated rx -180 ry 0 rz -60 deg; joints [-19.898, -51.3, 150.649, -80.002, -91.436, -8.316]
  MoveL 1357 to (445.86, -384.76, -5) mm, rotated rx 180 ry 0 rz -60 deg; joints [-19.357, -51.196, 148.981, -79.43, -91.236, -6.763]
  MoveC 1358 to (433.16, -397.46, -5) mm, rotated rx -180 ry 0 rz -60 deg; joints [-19.835, -51.091, 147.842, -79.885, -90.991, -5.756] to (420.46, -384.76, -5) mm, rotated rx -180 ry 0 rz -60 deg; joints [-18.844, -51.03, 147.294, -78.891, -91.011, -5.256]
  MoveL 1359 to (395.06, -384.76, -5) mm, rotated rx 180 ry 0 rz -30 deg; joints [-13.014, -51.124, 155.98, -43.881, -100.196, -9.566]
  MoveL 1360 to (318.86, -384.76, -5) mm, rotated rx -180 ry 0 rz 0 deg; joints [-1.265, -51.255, 155.308, -1.304, -103.18, -0.044]
  MoveC 1361 to (306.16, -397.46, -5) mm, rotated rx -180 ry 0 rz 0 deg; joints [-2.116, -51.32, 154.42, -2.169, -102.221, -0.219] to (293.46, -384.76, -5) mm, rotated rx -180 ry 0 rz 0 deg; joints [-1.227, -51.37, 153.582, -1.256, -101.339, 0.007]
  MoveL 1362 to (191.86, -384.76, -5) mm, rotated rx -180 ry 0 rz 0 deg; joints [-1.096, -50.992, 146.511, -1.103, -94.648, 0.166]
  MoveC 1363 to (179.16, -397.46, -5) mm, rotated rx -180 ry 0 rz 0 deg; joints [-1.836, -50.86, 145.584, -1.844, -93.853, 0.12] to (166.46, -384.76, -5) mm, rotated rx -180 ry 0 rz 0 deg; joints [-1.067, -50.73, 144.702, -1.073, -93.102, 0.198]
  MoveL 1364 to (90.26, -384.76, -5) mm, rotated rx 180 ry 0 rz 0 deg; joints [-0.989, -49.634, 139.177, -0.994, -88.674, 0.28]
  MoveL 1365 to (64.86, -384.76, -5) mm, rotated rx -180 ry 0 rz 0 deg; joints [-0.966, -49.178, 137.3, -0.971, -87.253, 0.304]
  MoveC 1366 to (61.14, -393.74, -5) mm, rotated rx -180 ry 0 rz 0 deg; joints [-1.438, -49.101, 137.009, -1.444, -87.039, 0.325] to (52.16, -397.46, -5) mm, rotated rx -180 ry 0 rz 0 deg; joints [-1.622, -48.925, 136.333, -1.629, -86.539, 0.346]
  MoveL 1367 to (52.16, -397.46, -5) mm, rotated rx -180 ry 0 rz 0 deg; joints [-1.622, -48.925, 136.333, -1.629, -86.539, 0.346]
  MoveC 1368 to (43.18, -393.74, -5) mm, rotated rx 180 ry 0 rz 0 deg; joints [-1.415, -48.751, 135.669, -1.422, -86.049, 0.349] to (39.46, -384.76, -5) mm, rotated rx 180 ry 0 rz 0 deg; joints [-0.944, -48.683, 135.405, -0.95, -85.853, 0.327]
  MoveL 1369 to (14.06, -384.76, -5) mm, rotated rx -180 ry 0 rz 0 deg; joints [-0.922, -48.151, 133.491, -0.931, -84.471, 0.348]
  MoveC 1370 to (13.61, -384.57, -5) mm, rotated rx -180 ry 0 rz 0 deg; joints [-0.913, -48.141, 133.457, -0.921, -84.447, 0.348] to (13.42, -384.12, -5) mm, rotated rx 180 ry 0 rz 0 deg; joints [-0.89, -48.137, 133.444, -0.898, -84.437, 0.346]
  MoveL 1371 to (13.42, -383.49, -5) mm, rotated rx 180 ry 0 rz 0 deg; joints [-0.857, -48.138, 133.444, -0.866, -84.437, 0.343]
  MoveC 1372 to (13.42, -383.04, -4.81) mm, rotated rx -180 ry 0 rz 0 deg; joints [-0.835, -48.153, 133.448, -0.843, -84.426, 0.341] to (13.42, -382.85, -4.37) mm, rotated rx -180 ry 0 rz 0 deg; joints [-0.825, -48.188, 133.455, -0.833, -84.398, 0.341]
  Set speed (500.0 mm/s)
  MoveL 1373 to (13.42, -382.85, 5) mm, rotated rx -180 ry 0 rz 0 deg; joints [-0.827, -48.916, 133.596, -0.836, -83.811, 0.35]
  MoveL 1374 to (12.15, -384.12, 5) mm, rotated rx 180 ry 0 rz 0 deg; joints [-0.891, -48.886, 133.498, -0.9, -83.743, 0.357]
  Set speed (25.4 mm/s)
  MoveL 1375 to (12.15, -384.12, 1) mm, rotated rx -180 ry 0 rz 0 deg; joints [-0.89, -48.576, 133.439, -0.899, -83.994, 0.353]
  MoveL 1376 to (12.15, -384.12, -7.71) mm, rotated rx -180 ry 0 rz 0 deg; joints [-0.888, -47.899, 133.305, -0.896, -84.537, 0.344]
  MoveC 1377 to (12.34, -384.12, -8.16) mm, rotated rx -180 ry 0 rz 0 deg; joints [-0.888, -47.868, 133.312, -0.896, -84.575, 0.344] to (12.79, -384.12, -8.35) mm, rotated rx -180 ry 0 rz 0 deg; joints [-0.888, -47.863, 133.343, -0.896, -84.611, 0.343]
  Set speed (50.8 mm/s)
  MoveL 1378 to (13.42, -384.12, -8.35) mm, rotated rx -180 ry 0 rz 0 deg; joints [-0.889, -47.877, 133.391, -0.897, -84.645, 0.342]
  MoveC 1379 to (13.87, -384.31, -8.35) mm, rotated rx -180 ry 0 rz 0 deg; joints [-0.899, -47.886, 133.425, -0.907, -84.669, 0.343] to (14.06, -384.76, -8.35) mm, rotated rx -180 ry 0 rz 0 deg; joints [-0.922, -47.89, 133.438, -0.93, -84.679, 0.345]
  MoveL 1380 to (14.06, -537.16, -8.35) mm, rotated rx -180 ry 0 rz 0 deg; joints [-8.597, -47.574, 132.467, -8.647, -84.082, 1.039]
  MoveL 1381 to (471.26, -537.16, -8.35) mm, rotated rx -180 ry 0 rz -30 deg; joints [-25.103, -50.488, 157.401, -56.136, -98.981, -13.309]
  MoveL 1382 to (471.26, -384.76, -8.35) mm, rotated rx -180 ry 0 rz -60 deg; joints [-19.899, -50.945, 150.579, -80.009, -91.485, -8.598]
  MoveL 1383 to (445.86, -384.76, -8.35) mm, rotated rx -180 ry 0 rz -60 deg; joints [-19.357, -50.853, 148.914, -79.436, -91.286, -7.034]
  MoveC 1384 to (433.16, -397.46, -8.35) mm, rotated rx -180 ry 0 rz -60 deg; joints [-19.835, -50.756, 147.777, -79.89, -91.038, -6.022] to (420.46, -384.76, -8.35) mm, rotated rx -180 ry 0 rz -60 deg; joints [-18.844, -50.699, 147.229, -78.896, -91.063, -5.518]
  MoveL 1385 to (395.06, -384.76, -8.35) mm, rotated rx 180 ry 0 rz -30 deg; joints [-13.014, -50.723, 155.901, -43.922, -100.43, -9.794]
  MoveL 1386 to (318.86, -384.76, -8.35) mm, rotated rx -180 ry 0 rz 0 deg; joints [-1.264, -50.86, 155.231, -1.304, -103.498, -0.051]
  MoveC 1387 to (306.16, -397.46, -8.35) mm, rotated rx -180 ry 0 rz 0 deg; joints [-2.115, -50.933, 154.345, -2.17, -102.533, -0.231] to (293.46, -384.76, -8.35) mm, rotated rx -180 ry 0 rz 0 deg; joints [-1.226, -50.99, 153.508, -1.256, -101.645, 0]
  MoveL 1388 to (191.86, -384.76, -8.35) mm, rotated rx -180 ry 0 rz 0 deg; joints [-1.095, -50.666, 146.447, -1.103, -94.911, 0.161]
  MoveC 1389 to (179.16, -397.46, -8.35) mm, rotated rx -180 ry 0 rz 0 deg; joints [-1.835, -50.539, 145.522, -1.844, -94.111, 0.112] to (166.46, -384.76, -8.35) mm, rotated rx 180 ry 0 rz 0 deg; joints [-1.066, -50.415, 144.641, -1.072, -93.355, 0.193]
  MoveL 1390 to (90.26, -384.76, -8.35) mm, rotated rx -180 ry 0 rz 0 deg; joints [-0.989, -49.348, 139.12, -0.993, -88.902, 0.276]
  MoveL 1391 to (64.86, -384.76, -8.35) mm, rotated rx -180 ry 0 rz 0 deg; joints [-0.965, -48.902, 137.245, -0.97, -87.474, 0.3]
  MoveC 1392 to (61.14, -393.74, -8.35) mm, rotated rx 180 ry 0 rz 0 deg; joints [-1.438, -48.826, 136.954, -1.443, -87.259, 0.319] to (52.16, -397.46, -8.35) mm, rotated rx -180 ry 0 rz 0 deg; joints [-1.621, -48.653, 136.278, -1.628, -86.757, 0.34]
  MoveL 1393 to (52.16, -397.46, -8.35) mm, rotated rx -180 ry 0 rz 0 deg; joints [-1.621, -48.653, 136.278, -1.628, -86.757, 0.34]
  MoveC 1394 to (43.18, -393.74, -8.35) mm, rotated rx -180 ry 0 rz 0 deg; joints [-1.414, -48.482, 135.615, -1.421, -86.265, 0.343] to (39.46, -384.76, -8.35) mm, rotated rx -180 ry 0 rz 0 deg; joints [-0.943, -48.415, 135.351, -0.949, -86.067, 0.323]
  MoveL 1395 to (14.06, -384.76, -8.35) mm, rotated rx 180 ry 0 rz 0 deg; joints [-0.922, -47.89, 133.438, -0.93, -84.679, 0.345]
  MoveC 1396 to (13.61, -384.57, -8.35) mm, rotated rx -180 ry 0 rz 0 deg; joints [-0.912, -47.881, 133.404, -0.92, -84.655, 0.344] to (13.42, -384.12, -8.35) mm, rotated rx -180 ry 0 rz 0 deg; joints [-0.889, -47.877, 133.391, -0.897, -84.645, 0.342]
  MoveL 1397 to (13.42, -383.49, -8.35) mm, rotated rx -180 ry 0 rz 0 deg; joints [-0.857, -47.877, 133.392, -0.864, -84.645, 0.34]
  MoveC 1398 to (13.42, -383.04, -8.16) mm, rotated rx -180 ry 0 rz 0 deg; joints [-0.834, -47.892, 133.395, -0.842, -84.634, 0.338] to (13.42, -382.85, -7.72) mm, rotated rx -180 ry 0 rz 0 deg; joints [-0.825, -47.927, 133.403, -0.832, -84.606, 0.338]
  Set speed (500.0 mm/s)
  MoveL 1399 to (13.42, -382.85, 6) mm, rotated rx 180 ry 0 rz 0 deg; joints [-0.828, -48.993, 133.611, -0.837, -83.748, 0.351]
  MoveL 1400 to (-13.42, -382.85, 6) mm, rotated rx -180 ry 0 rz 0 deg; joints [-0.808, -48.366, 131.562, -0.82, -82.327, 0.369]
  Set speed (25.4 mm/s)
  MoveL 1401 to (-13.42, -382.85, -4.36) mm, rotated rx -180 ry 0 rz 0 deg; joints [-0.806, -47.584, 131.41, -0.816, -82.956, 0.36]
  MoveC 1402 to (-13.42, -383.04, -4.81) mm, rotated rx 180 ry 0 rz 0 deg; joints [-0.815, -47.55, 131.403, -0.825, -82.983, 0.361] to (-13.42, -383.49, -5) mm, rotated rx 180 ry 0 rz 0 deg; joints [-0.837, -47.536, 131.399, -0.848, -82.994, 0.363]
  Set speed (50.8 mm/s)
  MoveL 1403 to (-13.42, -384.12, -5) mm, rotated rx -180 ry 0 rz 0 deg; joints [-0.869, -47.536, 131.399, -0.879, -82.994, 0.366]
  MoveC 1404 to (-13.61, -384.57, -5) mm, rotated rx -180 ry 0 rz 0 deg; joints [-0.891, -47.531, 131.384, -0.902, -82.984, 0.369] to (-14.06, -384.76, -5) mm, rotated rx -180 ry 0 rz 0 deg; joints [-0.9, -47.521, 131.349, -0.911, -82.96, 0.37]
  MoveL 1405 to (-39.46, -384.76, -5) mm, rotated rx -180 ry 0 rz 0 deg; joints [-0.88, -46.916, 129.392, -0.894, -81.607, 0.389]
  MoveC 1406 to (-52.16, -397.46, -5) mm, rotated rx 180 ry 0 rz 0 deg; joints [-1.48, -46.591, 128.384, -1.503, -80.926, 0.487] to (-64.86, -384.76, -5) mm, rotated rx -180 ry 0 rz 0 deg; joints [-0.862, -46.279, 127.413, -0.879, -80.265, 0.408]
  MoveL 1407 to (-90.26, -384.76, -5) mm, rotated rx -180 ry 0 rz 0 deg; joints [-0.844, -45.612, 125.411, -0.864, -78.93, 0.425]
  MoveL 1408 to (-166.46, -384.76, -5) mm, rotated rx -180 ry 0 rz 0 deg; joints [-0.795, -43.435, 119.254, -0.827, -74.95, 0.475]
  MoveC 1409 to (-179.16, -397.46, -5) mm, rotated rx -180 ry 0 rz 0 deg; joints [-1.337, -43.037, 118.183, -1.394, -74.281, 0.63] to (-191.86, -384.76, -5) mm, rotated rx -180 ry 0 rz 0 deg; joints [-0.779, -42.653, 117.146, -0.817, -73.625, 0.491]
  MoveL 1410 to (-293.46, -384.76, -5) mm, rotated rx -180 ry 0 rz 0 deg; joints [-0.724, -39.24, 108.391, -0.784, -68.283, 0.551]
  MoveC 1411 to (-306.16, -397.46, -5) mm, rotated rx -180 ry 0 rz 0 deg; joints [-1.22, -38.77, 107.235, -1.324, -67.6, 0.758] to (-318.86, -384.76, -5) mm, rotated rx -180 ry 0 rz 0 deg; joints [-0.711, -38.315, 106.109, -0.778, -66.926, 0.566]
  MoveL 1412 to (-395.06, -384.76, -5) mm, rotated rx -180 ry 0 rz 0 deg; joints [-0.676, -35.353, 98.994, -0.765, -62.774, 0.612]
  MoveL 1413 to (-420.46, -384.76, -5) mm, rotated rx 180 ry 0 rz 0 deg; joints [-0.665, -34.299, 96.52, -0.762, -61.353, 0.628]
  MoveC 1414 to (-433.16, -397.46, -5) mm, rotated rx 180 ry 0 rz 0 deg; joints [-1.121, -33.747, 95.24, -1.291, -60.63, 0.889] to (-445.86, -384.76, -5) mm, rotated rx -180 ry 0 rz 0 deg; joints [-0.654, -33.208, 93.986, -0.761, -59.91, 0.644]
  MoveL 1415 to (-471.26, -384.76, -5) mm, rotated rx 180 ry 0 rz 0 deg; joints [-0.644, -32.079, 91.388, -0.76, -58.441, 0.66]
  MoveL 1416 to (-471.26, -537.16, -5) mm, rotated rx -180 ry 0 rz 0 deg; joints [-6.034, -31.644, 90.453, -7.113, -58.134, 3.95]
  MoveL 1417 to (-14.06, -537.16, -5) mm, rotated rx -180 ry 0 rz 0 deg; joints [-8.392, -47.19, 130.39, -8.47, -82.403, 1.272]
  MoveL 1418 to (-14.06, -384.76, -5) mm, rotated rx -180 ry 0 rz 0 deg; joints [-0.9, -47.521, 131.349, -0.911, -82.96, 0.37]
  MoveC 1419 to (-13.87, -384.31, -5) mm, rotated rx 180 ry 0 rz 0 deg; joints [-0.878, -47.525, 131.364, -0.888, -82.97, 0.368] to (-13.42, -384.12, -5) mm, rotated rx -180 ry 0 rz 0 deg; joints [-0.869, -47.536, 131.399, -0.879, -82.994, 0.366]
  MoveL 1420 to (-12.79, -384.12, -5) mm, rotated rx 180 ry 0 rz 0 deg; joints [-0.869, -47.55, 131.447, -0.88, -83.028, 0.366]
  MoveC 1421 to (-12.34, -384.12, -4.81) mm, rotated rx -180 ry 0 rz 0 deg; joints [-0.87, -47.575, 131.484, -0.88, -83.041, 0.366] to (-12.15, -384.12, -4.37) mm, rotated rx -180 ry 0 rz 0 deg; joints [-0.87, -47.613, 131.505, -0.881, -83.024, 0.366]
  Set speed (500.0 mm/s)
  MoveL 1422 to (-12.15, -384.12, 5) mm, rotated rx 180 ry 0 rz 0 deg; joints [-0.872, -48.32, 131.643, -0.884, -82.454, 0.375]
  MoveL 1423 to (-13.42, -382.85, 5) mm, rotated rx 180 ry 0 rz 0 deg; joints [-0.808, -48.291, 131.548, -0.819, -82.388, 0.369]
  Set speed (25.4 mm/s)
  MoveL 1424 to (-13.42, -382.85, 1) mm, rotated rx -180 ry 0 rz 0 deg; joints [-0.807, -47.989, 131.49, -0.818, -82.632, 0.365]
  MoveL 1425 to (-13.42, -382.85, -7.72) mm, rotated rx -180 ry 0 rz 0 deg; joints [-0.805, -47.332, 131.358, -0.815, -83.158, 0.357]
  MoveC 1426 to (-13.42, -383.04, -8.16) mm, rotated rx 180 ry 0 rz 0 deg; joints [-0.814, -47.298, 131.351, -0.824, -83.185, 0.358] to (-13.42, -383.49, -8.35) mm, rotated rx 180 ry 0 rz 0 deg; joints [-0.837, -47.283, 131.348, -0.847, -83.196, 0.36]
  Set speed (50.8 mm/s)
  MoveL 1427 to (-13.42, -384.12, -8.35) mm, rotated rx 180 ry 0 rz 0 deg; joints [-0.868, -47.283, 131.347, -0.878, -83.195, 0.363]
  MoveC 1428 to (-13.61, -384.57, -8.35) mm, rotated rx -180 ry 0 rz 0 deg; joints [-0.89, -47.278, 131.332, -0.901, -83.185, 0.366] to (-14.06, -384.76, -8.35) mm, rotated rx 180 ry 0 rz 0 deg; joints [-0.899, -47.268, 131.298, -0.91, -83.161, 0.367]
  MoveL 1429 to (-39.46, -384.76, -8.35) mm, rotated rx 180 ry 0 rz 0 deg; joints [-0.88, -46.67, 129.341, -0.893, -81.803, 0.386]
  MoveC 1430 to (-52.16, -397.46, -8.35) mm, rotated rx -180 ry 0 rz 0 deg; joints [-1.479, -46.348, 128.334, -1.501, -81.119, 0.482] to (-64.86, -384.76, -8.35) mm, rotated rx 180 ry 0 rz 0 deg; joints [-0.861, -46.04, 127.363, -0.877, -80.455, 0.405]
  MoveL 1431 to (-90.26, -384.76, -8.35) mm, rotated rx -180 ry 0 rz 0 deg; joints [-0.843, -45.379, 125.362, -0.863, -79.115, 0.422]
  MoveL 1432 to (-166.46, -384.76, -8.35) mm, rotated rx 180 ry 0 rz 0 deg; joints [-0.794, -43.219, 119.207, -0.826, -75.12, 0.472]
  MoveC 1433 to (-179.16, -397.46, -8.35) mm, rotated rx -180 ry 0 rz 0 deg; joints [-1.337, -42.822, 118.137, -1.392, -74.449, 0.625] to (-191.86, -384.76, -8.35) mm, rotated rx 180 ry 0 rz 0 deg; joints [-0.779, -42.441, 117.1, -0.815, -73.791, 0.488]
  MoveL 1434 to (-293.46, -384.76, -8.35) mm, rotated rx 180 ry 0 rz 0 deg; joints [-0.723, -39.046, 108.346, -0.782, -68.432, 0.549]
  MoveC 1435 to (-306.16, -397.46, -8.35) mm, rotated rx -180 ry 0 rz 0 deg; joints [-1.219, -38.578, 107.191, -1.322, -67.748, 0.754] to (-318.86, -384.76, -8.35) mm, rotated rx -180 ry 0 rz 0 deg; joints [-0.711, -38.125, 106.065, -0.776, -67.073, 0.564]
  MoveL 1436 to (-395.06, -384.76, -8.35) mm, rotated rx -180 ry 0 rz 0 deg; joints [-0.675, -35.173, 98.95, -0.763, -62.91, 0.61]
  MoveL 1437 to (-420.46, -384.76, -8.35) mm, rotated rx 180 ry 0 rz 0 deg; joints [-0.664, -34.122, 96.476, -0.761, -61.486, 0.625]
  MoveC 1438 to (-433.16, -397.46, -8.35) mm, rotated rx -180 ry 0 rz 0 deg; joints [-1.121, -33.571, 95.196, -1.289, -60.761, 0.885] to (-445.86, -384.76, -8.35) mm, rotated rx -180 ry 0 rz 0 deg; joints [-0.654, -33.034, 93.942, -0.759, -60.04, 0.641]
  MoveL 1439 to (-471.26, -384.76, -8.35) mm, rotated rx -180 ry 0 rz 0 deg; joints [-0.643, -31.908, 91.343, -0.759, -58.568, 0.658]
  MoveL 1440 to (-471.26, -537.16, -8.35) mm, rotated rx -180 ry 0 rz 0 deg; joints [-6.033, -31.474, 90.409, -7.103, -58.258, 3.931]
  MoveL 1441 to (-14.06, -537.16, -8.35) mm, rotated rx 180 ry 0 rz 0 deg; joints [-8.391, -46.941, 130.339, -8.465, -82.6, 1.242]
  MoveL 1442 to (-14.06, -384.76, -8.35) mm, rotated rx 180 ry 0 rz 0 deg; joints [-0.899, -47.268, 131.298, -0.91, -83.161, 0.367]
  MoveC 1443 to (-13.87, -384.31, -8.35) mm, rotated rx 180 ry 0 rz 0 deg; joints [-0.877, -47.272, 131.312, -0.887, -83.171, 0.364] to (-13.42, -384.12, -8.35) mm, rotated rx 180 ry 0 rz 0 deg; joints [-0.868, -47.283, 131.347, -0.878, -83.195, 0.363]
  MoveL 1444 to (-12.79, -384.12, -8.35) mm, rotated rx -180 ry 0 rz 0 deg; joints [-0.869, -47.297, 131.396, -0.879, -83.23, 0.363]
  MoveC 1445 to (-12.34, -384.12, -8.16) mm, rotated rx -180 ry 0 rz 0 deg; joints [-0.869, -47.322, 131.433, -0.879, -83.243, 0.363] to (-12.15, -384.12, -7.72) mm, rotated rx -180 ry 0 rz 0 deg; joints [-0.869, -47.36, 131.454, -0.879, -83.226, 0.363]
  Set speed (500.0 mm/s)
  MoveL 1446 to (-12.15, -384.12, 6) mm, rotated rx 180 ry 0 rz 0 deg; joints [-0.872, -48.396, 131.658, -0.884, -82.393, 0.376]
  MoveL 1447 to (-52.79, 196.51, 6) mm, rotated rx -180 ry 0 rz 0 deg; joints [25.227, -44.064, 118.453, 26.169, -75.047, -6.544]
  Set speed (25.4 mm/s)
  MoveL 1448 to (-52.79, 196.51, -4.37) mm, rotated rx -180 ry 0 rz 0 deg; joints [25.232, -43.402, 118.318, 26.113, -75.519, -6.306]
  MoveC 1449 to (-52.79, 196.7, -4.81) mm, rotated rx 180 ry 0 rz 0 deg; joints [25.239, -43.371, 118.305, 26.119, -75.537, -6.299] to (-52.79, 197.15, -5) mm, rotated rx 180 ry 0 rz 0 deg; joints [25.257, -43.354, 118.287, 26.137, -75.538, -6.304]
  Set speed (50.8 mm/s)
  MoveL 1450 to (-52.79, 197.78, -5) mm, rotated rx -180 ry 0 rz 0 deg; joints [25.282, -43.346, 118.264, 26.165, -75.528, -6.317]
  MoveC 1451 to (-52.61, 198.23, -5) mm, rotated rx -180 ry 0 rz 0 deg; joints [25.303, -43.345, 118.262, 26.186, -75.529, -6.322] to (-52.16, 198.42, -5) mm, rotated rx -180 ry 0 rz 0 deg; joints [25.319, -43.356, 118.289, 26.2, -75.546, -6.319]
  MoveL 1452 to (-14.06, 198.42, -5) mm, rotated rx 180 ry 0 rz 0 deg; joints [26.044, -44.401, 121.114, 26.75, -77.218, -5.666]
  MoveL 1453 to (-14.06, 350.82, -5) mm, rotated rx 180 ry 0 rz 0 deg; joints [31.819, -42.213, 115.002, 33.148, -74.58, -9.04]
  MoveL 1454 to (-39.46, 350.82, -5) mm, rotated rx -180 ry 0 rz 0 deg; joints [31.264, -41.488, 113.152, 32.754, -73.543, -9.528]
  MoveC 1455 to (-52.16, 338.12, -5) mm, rotated rx -180 ry 0 rz 0 deg; joints [30.543, -41.328, 112.772, 32.048, -73.235, -9.45] to (-64.86, 350.82, -5) mm, rotated rx 180 ry 0 rz 0 deg; joints [30.726, -40.738, 111.265, 32.387, -72.491, -10.015]
  MoveL 1456 to (-90.26, 350.82, -5) mm, rotated rx 180 ry 0 rz 0 deg; joints [30.205, -39.964, 109.342, 32.048, -71.424, -10.5]
  MoveL 1457 to (-166.46, 350.82, -5) mm, rotated rx 180 ry 0 rz 0 deg; joints [28.733, -37.486, 103.33, 31.193, -68.121, -11.965]
  MoveC 1458 to (-179.16, 338.12, -5) mm, rotated rx -180 ry 0 rz 0 deg; joints [28.074, -37.276, 102.851, 30.553, -67.75, -11.864] to (-191.86, 350.82, -5) mm, rotated rx -180 ry 0 rz 0 deg; joints [28.272, -36.605, 101.239, 30.963, -66.984, -12.462]
  MoveL 1459 to (-293.46, 350.82, -5) mm, rotated rx -180 ry 0 rz 0 deg; joints [26.554, -32.78, 92.362, 30.338, -62.228, -14.547]
  MoveC 1460 to (-306.16, 338.12, -5) mm, rotated rx 180 ry 0 rz 0 deg; joints [25.948, -32.511, 91.765, 29.762, -61.79, -14.431] to (-318.86, 350.82, -5) mm, rotated rx 180 ry 0 rz 0 deg; joints [26.154, -31.739, 89.996, 30.261, -60.98, -15.105]
  MoveL 1461 to (-395.06, 350.82, -5) mm, rotated rx -180 ry 0 rz 0 deg; joints [25.02, -28.376, 82.458, 30.254, -57.055, -16.921]
  MoveL 1462 to (-420.46, 350.82, -5) mm, rotated rx 180 ry 0 rz 0 deg; joints [24.662, -27.162, 79.774, 30.338, -55.678, -17.59]
  MoveC 1463 to (-433.16, 338.12, -5) mm, rotated rx 180 ry 0 rz 0 deg; joints [24.103, -26.813, 79.019, 29.832, -55.156, -17.479] to (-445.86, 350.82, -5) mm, rotated rx 180 ry 0 rz 0 deg; joints [24.314, -25.894, 76.988, 30.472, -54.26, -18.302]
  MoveL 1464 to (-471.26, 350.82, -5) mm, rotated rx -180 ry 0 rz 0 deg; joints [23.974, -24.566, 74.087, 30.665, -52.795, -19.065]
  MoveL 1465 to (-471.26, 198.42, -5) mm, rotated rx -180 ry 0 rz 0 deg; joints [19.302, -27.611, 80.919, 23.844, -54.827, -13.707]
  MoveL 1466 to (-445.86, 198.42, -5) mm, rotated rx 180 ry 0 rz 0 deg; joints [19.587, -28.848, 83.667, 23.762, -56.277, -13.153]
  MoveL 1467 to (-52.16, 198.42, -5) mm, rotated rx -180 ry 0 rz 0 deg; joints [25.319, -43.356, 118.289, 26.2, -75.546, -6.319]
  MoveC 1468 to (-51.71, 198.23, -5) mm, rotated rx -180 ry 0 rz 0 deg; joints [25.32, -43.371, 118.33, 26.199, -75.569, -6.307] to (-51.52, 197.78, -5) mm, rotated rx -180 ry 0 rz 0 deg; joints [25.305, -43.382, 118.359, 26.182, -75.584, -6.295]
  MoveL 1469 to (-51.52, 197.15, -5) mm, rotated rx -180 ry 0 rz 0 deg; joints [25.281, -43.39, 118.382, 26.155, -75.594, -6.283]
  MoveC 1470 to (-51.52, 196.7, -4.81) mm, rotated rx -180 ry 0 rz 0 deg; joints [25.263, -43.407, 118.4, 26.136, -75.593, -6.278] to (-51.52, 196.52, -4.37) mm, rotated rx -180 ry 0 rz 0 deg; joints [25.255, -43.438, 118.413, 26.131, -75.576, -6.285]
  Set speed (500.0 mm/s)
  MoveL 1471 to (-51.52, 196.51, 5) mm, rotated rx -180 ry 0 rz 0 deg; joints [25.251, -44.036, 118.536, 26.181, -75.148, -6.5]
  MoveL 1472 to (-52.79, 196.51, 5) mm, rotated rx -180 ry 0 rz 0 deg; joints [25.227, -44, 118.44, 26.164, -75.093, -6.521]
  Set speed (25.4 mm/s)
  MoveL 1473 to (-52.79, 196.52, 1) mm, rotated rx -180 ry 0 rz 0 deg; joints [25.229, -43.745, 118.389, 26.142, -75.276, -6.429]
  MoveL 1474 to (-52.79, 196.51, -7.71) mm, rotated rx -180 ry 0 rz 0 deg; joints [25.233, -43.188, 118.272, 26.096, -75.671, -6.23]
  MoveC 1475 to (-52.79, 196.7, -8.16) mm, rotated rx -180 ry 0 rz 0 deg; joints [25.241, -43.157, 118.259, 26.102, -75.688, -6.223] to (-52.79, 197.15, -8.35) mm, rotated rx -180 ry 0 rz 0 deg; joints [25.259, -43.14, 118.241, 26.12, -75.689, -6.228]
  Set speed (50.8 mm/s)
  MoveL 1476 to (-52.79, 197.78, -8.35) mm, rotated rx -180 ry 0 rz 0 deg; joints [25.284, -43.132, 118.218, 26.147, -75.679, -6.24]
  MoveC 1477 to (-52.61, 198.23, -8.35) mm, rotated rx 180 ry 0 rz 0 deg; joints [25.305, -43.131, 118.216, 26.169, -75.68, -6.246] to (-52.16, 198.42, -8.35) mm, rotated rx 180 ry 0 rz 0 deg; joints [25.32, -43.141, 118.243, 26.183, -75.697, -6.242]
  MoveL 1478 to (-14.06, 198.42, -8.35) mm, rotated rx 180 ry 0 rz 0 deg; joints [26.046, -44.18, 121.067, 26.734, -77.374, -5.586]
  MoveL 1479 to (-14.06, 350.82, -8.35) mm, rotated rx -180 ry 0 rz 0 deg; joints [31.821, -42.006, 114.957, 33.125, -74.715, -8.948]
  MoveL 1480 to (-39.46, 350.82, -8.35) mm, rotated rx 180 ry 0 rz 0 deg; joints [31.266, -41.285, 113.107, 32.73, -73.677, -9.44]
  MoveC 1481 to (-52.16, 338.12, -8.35) mm, rotated rx 180 ry 0 rz 0 deg; joints [30.545, -41.126, 112.728, 32.024, -73.369, -9.364] to (-64.86, 350.82, -8.35) mm, rotated rx -180 ry 0 rz 0 deg; joints [30.728, -40.539, 111.221, 32.363, -72.622, -9.928]
  MoveL 1482 to (-90.26, 350.82, -8.35) mm, rotated rx 180 ry 0 rz 0 deg; joints [30.207, -39.768, 109.298, 32.022, -71.553, -10.416]
  MoveL 1483 to (-166.46, 350.82, -8.35) mm, rotated rx 180 ry 0 rz 0 deg; joints [28.735, -37.3, 103.287, 31.165, -68.243, -11.886]
  MoveC 1484 to (-179.16, 338.12, -8.35) mm, rotated rx -180 ry 0 rz 0 deg; joints [28.075, -37.091, 102.807, 30.526, -67.872, -11.786] to (-191.86, 350.82, -8.35) mm, rotated rx 180 ry 0 rz 0 deg; joints [28.273, -36.422, 101.195, 30.935, -67.104, -12.385]
  MoveL 1485 to (-293.46, 350.82, -8.35) mm, rotated rx 180 ry 0 rz 0 deg; joints [26.555, -32.608, 92.318, 30.306, -62.339, -14.474]
  MoveC 1486 to (-306.16, 338.12, -8.35) mm, rotated rx -180 ry 0 rz 0 deg; joints [25.949, -32.34, 91.721, 29.73, -61.901, -14.36] to (-318.86, 350.82, -8.35) mm, rotated rx -180 ry 0 rz 0 deg; joints [26.155, -31.57, 89.951, 30.228, -61.088, -15.033]
  MoveL 1487 to (-395.06, 350.82, -8.35) mm, rotated rx -180 ry 0 rz 0 deg; joints [25.021, -28.213, 82.412, 30.218, -57.157, -16.852]
  MoveL 1488 to (-420.46, 350.82, -8.35) mm, rotated rx -180 ry 0 rz 0 deg; joints [24.663, -27.001, 79.727, 30.3, -55.777, -17.521]
  MoveC 1489 to (-433.16, 338.12, -8.35) mm, rotated rx -180 ry 0 rz 0 deg; joints [24.104, -26.653, 78.972, 29.794, -55.255, -17.411] to (-445.86, 350.82, -8.35) mm, rotated rx -180 ry 0 rz 0 deg; joints [24.315, -25.735, 76.94, 30.433, -54.357, -18.233]
  MoveL 1490 to (-471.26, 350.82, -8.35) mm, rotated rx 180 ry 0 rz 0 deg; joints [23.976, -24.409, 74.038, 30.624, -52.89, -18.996]
  MoveL 1491 to (-471.26, 198.42, -8.35) mm, rotated rx -180 ry 0 rz 0 deg; joints [19.303, -27.449, 80.872, 23.813, -54.933, -13.651]
  MoveL 1492 to (-445.86, 198.42, -8.35) mm, rotated rx -180 ry 0 rz 0 deg; joints [19.588, -28.685, 83.622, 23.731, -56.385, -13.097]
  MoveL 1493 to (-52.16, 198.42, -8.35) mm, rotated rx 180 ry 0 rz 0 deg; joints [25.32, -43.141, 118.243, 26.183, -75.697, -6.242]
  MoveC 1494 to (-51.71, 198.23, -8.35) mm, rotated rx -180 ry 0 rz 0 deg; joints [25.321, -43.156, 118.284, 26.181, -75.72, -6.231] to (-51.52, 197.78, -8.35) mm, rotated rx 180 ry 0 rz 0 deg; joints [25.307, -43.167, 118.314, 26.165, -75.736, -6.219]
  MoveL 1495 to (-51.52, 197.15, -8.35) mm, rotated rx -180 ry 0 rz 0 deg; joints [25.282, -43.175, 118.336, 26.137, -75.746, -6.206]
  MoveC 1496 to (-51.52, 196.7, -8.16) mm, rotated rx -180 ry 0 rz 0 deg; joints [25.264, -43.193, 118.354, 26.119, -75.745, -6.202] to (-51.52, 196.52, -7.72) mm, rotated rx -180 ry 0 rz 0 deg; joints [25.257, -43.224, 118.367, 26.113, -75.727, -6.208]
  Set speed (500.0 mm/s)
  MoveL 1497 to (-51.52, 196.51, 6) mm, rotated rx 180 ry 0 rz 0 deg; joints [25.251, -44.1, 118.549, 26.187, -75.103, -6.523]
  MoveL 1498 to (18.41, 196.52, 6) mm, rotated rx -180 ry 0 rz 0 deg; joints [26.61, -46.016, 123.686, 27.232, -78.127, -5.336]
  Set speed (25.4 mm/s)
  MoveL 1499 to (18.41, 196.51, -4.36) mm, rotated rx -180 ry 0 rz 0 deg; joints [26.615, -45.313, 123.545, 27.184, -78.628, -5.074]
  MoveC 1500 to (18.41, 196.7, -4.81) mm, rotated rx -180 ry 0 rz 0 deg; joints [26.623, -45.28, 123.532, 27.19, -78.646, -5.067] to (18.41, 197.15, -5) mm, rotated rx 180 ry 0 rz 0 deg; joints [26.641, -45.262, 123.514, 27.209, -78.648, -5.07]
  Set speed (50.8 mm/s)
  MoveL 1501 to (18.41, 197.78, -5) mm, rotated rx 180 ry 0 rz 0 deg; joints [26.667, -45.255, 123.491, 27.236, -78.636, -5.082]
  MoveC 1502 to (18.6, 198.23, -5) mm, rotated rx -180 ry 0 rz 0 deg; joints [26.689, -45.254, 123.488, 27.259, -78.637, -5.087] to (19.04, 198.42, -5) mm, rotated rx -180 ry 0 rz 0 deg; joints [26.706, -45.263, 123.514, 27.275, -78.653, -5.083]
  MoveL 1503 to (39.46, 198.42, -5) mm, rotated rx -180 ry 0 rz 0 deg; joints [27.13, -45.773, 124.969, 27.621, -79.53, -4.714]
  MoveL 1504 to (471.26, 198.42, -5) mm, rotated rx -180 ry 0 rz 0 deg; joints [40.1, -52.03, 151.771, 40.41, -96.573, 6.57]
  MoveL 1505 to (471.26, 350.82, -5) mm, rotated rx -180 ry 0 rz 0 deg; joints [46.916, -51.424, 144.401, 46.917, -91.164, 2.446]
  MoveL 1506 to (445.86, 350.82, -5) mm, rotated rx -180 ry 0 rz 0 deg; joints [45.853, -51.173, 143.136, 45.844, -90.497, 1.68]
  MoveC 1507 to (433.16, 338.12, -5) mm, rotated rx -180 ry 0 rz 0 deg; joints [44.823, -51.152, 143.139, 44.815, -90.54, 1.673] to (420.46, 350.82, -5) mm, rotated rx -180 ry 0 rz 0 deg; joints [44.827, -50.895, 141.838, 44.816, -89.799, 0.937]
  MoveL 1508 to (395.06, 350.82, -5) mm, rotated rx -180 ry 0 rz 0 deg; joints [43.836, -50.59, 140.51, 43.833, -89.073, 0.217]
  MoveL 1509 to (318.86, 350.82, -5) mm, rotated rx -180 ry 0 rz 0 deg; joints [41.067, -49.516, 136.343, 41.138, -86.739, -1.815]
  MoveC 1510 to (306.16, 338.12, -5) mm, rotated rx -180 ry 0 rz 0 deg; joints [40.128, -49.469, 136.236, 40.2, -86.659, -1.814] to (293.46, 350.82, -5) mm, rotated rx -180 ry 0 rz 0 deg; joints [40.206, -49.106, 134.894, 40.32, -85.916, -2.452]
  MoveL 1511 to (191.86, 350.82, -5) mm, rotated rx 180 ry 0 rz 0 deg; joints [37.049, -47.216, 128.808, 37.421, -82.432, -4.826]
  MoveC 1512 to (179.16, 338.12, -5) mm, rotated rx -180 ry 0 rz 0 deg; joints [36.195, -47.134, 128.601, 36.573, -82.256, -4.801] to (166.46, 350.82, -5) mm, rotated rx 180 ry 0 rz 0 deg; joints [36.326, -46.683, 127.214, 36.784, -81.517, -5.382]
  MoveL 1513 to (90.26, 350.82, -5) mm, rotated rx 180 ry 0 rz 0 deg; joints [34.294, -44.942, 122.252, 35.064, -78.681, -6.979]
  MoveL 1514 to (64.86, 350.82, -5) mm, rotated rx 180 ry 0 rz 0 deg; joints [33.661, -44.314, 120.536, 34.553, -77.705, -7.491]
  MoveC 1515 to (61.14, 341.84, -5) mm, rotated rx -180 ry 0 rz 0 deg; joints [33.238, -44.361, 120.686, 34.111, -77.733, -7.348] to (52.16, 338.12, -5) mm, rotated rx 180 ry 0 rz 0 deg; joints [32.884, -44.191, 120.234, 33.786, -77.452, -7.436]
  MoveL 1516 to (52.16, 338.12, -5) mm, rotated rx 180 ry 0 rz 0 deg; joints [32.884, -44.191, 120.234, 33.786, -77.452, -7.436]
  MoveC 1517 to (43.18, 341.84, -5) mm, rotated rx -180 ry 0 rz 0 deg; joints [32.807, -43.902, 119.449, 33.771, -77.029, -7.703] to (39.46, 350.82, -5) mm, rotated rx -180 ry 0 rz 0 deg; joints [33.048, -43.663, 118.79, 34.07, -76.714, -7.996]
  MoveL 1518 to (14.06, 350.82, -5) mm, rotated rx 180 ry 0 rz 0 deg; joints [32.454, -42.988, 117.01, 33.617, -75.709, -8.494]
  MoveL 1519 to (14.06, 198.42, -5) mm, rotated rx -180 ry 0 rz 0 deg; joints [26.604, -45.136, 123.155, 27.193, -78.437, -5.172]
  MoveL 1520 to (19.04, 198.42, -5) mm, rotated rx -180 ry 0 rz 0 deg; joints [26.706, -45.263, 123.514, 27.275, -78.653, -5.083]
  MoveC 1521 to (19.49, 198.23, -5) mm, rotated rx -180 ry 0 rz 0 deg; joints [26.708, -45.277, 123.553, 27.274, -78.675, -5.071] to (19.68, 197.79, -5) mm, rotated rx -180 ry 0 rz 0 deg; joints [26.693, -45.287, 123.582, 27.257, -78.691, -5.06]
  MoveL 1522 to (19.68, 197.15, -5) mm, rotated rx -180 ry 0 rz 0 deg; joints [26.667, -45.295, 123.605, 27.23, -78.702, -5.048]
  MoveC 1523 to (19.68, 196.7, -4.81) mm, rotated rx -180 ry 0 rz 0 deg; joints [26.649, -45.313, 123.623, 27.211, -78.701, -5.044] to (19.68, 196.52, -4.37) mm, rotated rx 180 ry 0 rz 0 deg; joints [26.641, -45.345, 123.636, 27.205, -78.683, -5.052]
  Set speed (500.0 mm/s)
  MoveL 1524 to (19.68, 196.51, 5) mm, rotated rx -180 ry 0 rz 0 deg; joints [26.636, -45.981, 123.764, 27.248, -78.23, -5.288]
  MoveL 1525 to (18.41, 196.51, 5) mm, rotated rx -180 ry 0 rz 0 deg; joints [26.61, -45.948, 123.672, 27.227, -78.176, -5.311]
  Set speed (25.4 mm/s)
  MoveL 1526 to (18.41, 196.51, 1) mm, rotated rx -180 ry 0 rz 0 deg; joints [26.612, -45.677, 123.619, 27.208, -78.37, -5.209]
  MoveL 1527 to (18.41, 196.51, -7.71) mm, rotated rx 180 ry 0 rz 0 deg; joints [26.617, -45.085, 123.498, 27.169, -78.789, -4.991]
  MoveC 1528 to (18.41, 196.7, -8.16) mm, rotated rx -180 ry 0 rz 0 deg; joints [26.625, -45.053, 123.485, 27.175, -78.807, -4.983] to (18.41, 197.15, -8.35) mm, rotated rx 180 ry 0 rz 0 deg; joints [26.643, -45.035, 123.466, 27.194, -78.808, -4.987]
  Set speed (50.8 mm/s)
  MoveL 1529 to (18.41, 197.78, -8.35) mm, rotated rx -180 ry 0 rz 0 deg; joints [26.669, -45.027, 123.443, 27.222, -78.797, -4.999]
  MoveC 1530 to (18.6, 198.23, -8.35) mm, rotated rx -180 ry 0 rz 0 deg; joints [26.691, -45.027, 123.441, 27.244, -78.797, -5.004] to (19.04, 198.42, -8.35) mm, rotated rx -180 ry 0 rz 0 deg; joints [26.708, -45.036, 123.466, 27.26, -78.813, -4.999]
  MoveL 1531 to (39.46, 198.42, -8.35) mm, rotated rx -180 ry 0 rz 0 deg; joints [27.132, -45.542, 124.921, 27.607, -79.693, -4.628]
  MoveL 1532 to (471.26, 198.42, -8.35) mm, rotated rx -180 ry 0 rz 0 deg; joints [40.103, -51.665, 151.701, 40.435, -96.796, 6.763]
  MoveL 1533 to (471.26, 350.82, -8.35) mm, rotated rx -180 ry 0 rz 0 deg; joints [46.918, -51.111, 144.341, 46.924, -91.337, 2.631]
  MoveL 1534 to (445.86, 350.82, -8.35) mm, rotated rx -180 ry 0 rz 0 deg; joints [45.855, -50.868, 143.076, 45.848, -90.669, 1.857]
  MoveC 1535 to (433.16, 338.12, -8.35) mm, rotated rx -180 ry 0 rz 0 deg; joints [44.826, -50.846, 143.08, 44.82, -90.715, 1.847] to (420.46, 350.82, -8.35) mm, rotated rx 180 ry 0 rz 0 deg; joints [44.829, -50.597, 141.78, 44.819, -89.97, 1.107]
  MoveL 1536 to (395.06, 350.82, -8.35) mm, rotated rx -180 ry 0 rz 0 deg; joints [43.839, -50.298, 140.453, 43.833, -89.242, 0.379]
  MoveL 1537 to (318.86, 350.82, -8.35) mm, rotated rx -180 ry 0 rz 0 deg; joints [41.069, -49.243, 136.289, 41.132, -86.904, -1.671]
  MoveC 1538 to (306.16, 338.12, -8.35) mm, rotated rx -180 ry 0 rz 0 deg; joints [40.13, -49.197, 136.182, 40.195, -86.826, -1.673] to (293.46, 350.82, -8.35) mm, rotated rx 180 ry 0 rz 0 deg; joints [40.209, -48.84, 134.841, 40.313, -86.079, -2.313]
  MoveL 1539 to (191.86, 350.82, -8.35) mm, rotated rx -180 ry 0 rz 0 deg; joints [37.052, -46.973, 128.759, 37.408, -82.586, -4.707]
  MoveC 1540 to (179.16, 338.12, -8.35) mm, rotated rx 180 ry 0 rz 0 deg; joints [36.197, -46.891, 128.552, 36.56, -82.412, -4.684] to (166.46, 350.82, -8.35) mm, rotated rx 180 ry 0 rz 0 deg; joints [36.328, -46.445, 127.165, 36.769, -81.67, -5.267]
  MoveL 1541 to (90.26, 350.82, -8.35) mm, rotated rx -180 ry 0 rz 0 deg; joints [34.296, -44.717, 122.205, 35.046, -78.826, -6.875]
  MoveL 1542 to (64.86, 350.82, -8.35) mm, rotated rx 180 ry 0 rz 0 deg; joints [33.663, -44.094, 120.49, 34.533, -77.848, -7.391]
  MoveC 1543 to (61.14, 341.84, -8.35) mm, rotated rx 180 ry 0 rz 0 deg; joints [33.24, -44.141, 120.639, 34.092, -77.877, -7.248] to (52.16, 338.12, -8.35) mm, rotated rx 180 ry 0 rz 0 deg; joints [32.885, -43.972, 120.188, 33.767, -77.596, -7.338]
  MoveL 1544 to (52.16, 338.12, -8.35) mm, rotated rx 180 ry 0 rz 0 deg; joints [32.885, -43.972, 120.188, 33.767, -77.596, -7.338]
  MoveC 1545 to (43.18, 341.84, -8.35) mm, rotated rx 180 ry 0 rz 0 deg; joints [32.809, -43.685, 119.403, 33.751, -77.171, -7.606] to (39.46, 350.82, -8.35) mm, rotated rx 180 ry 0 rz 0 deg; joints [33.05, -43.447, 118.744, 34.05, -76.855, -7.899]
  MoveL 1546 to (14.06, 350.82, -8.35) mm, rotated rx -180 ry 0 rz 0 deg; joints [32.456, -42.777, 116.965, 33.595, -75.848, -8.4]
  MoveL 1547 to (14.06, 198.42, -8.35) mm, rotated rx -180 ry 0 rz 0 deg; joints [26.606, -44.909, 123.108, 27.178, -78.597, -5.089]
  MoveL 1548 to (19.04, 198.42, -8.35) mm, rotated rx -180 ry 0 rz 0 deg; joints [26.708, -45.036, 123.466, 27.26, -78.813, -4.999]
  MoveC 1549 to (19.49, 198.23, -8.35) mm, rotated rx -180 ry 0 rz 0 deg; joints [26.709, -45.049, 123.505, 27.259, -78.836, -4.987] to (19.68, 197.78, -8.35) mm, rotated rx -180 ry 0 rz 0 deg; joints [26.695, -45.059, 123.534, 27.243, -78.852, -4.976]
  MoveL 1550 to (19.68, 197.15, -8.35) mm, rotated rx -180 ry 0 rz 0 deg; joints [26.669, -45.067, 123.557, 27.215, -78.863, -4.964]
  MoveC 1551 to (19.68, 196.7, -8.16) mm, rotated rx 180 ry 0 rz 0 deg; joints [26.651, -45.085, 123.576, 27.196, -78.862, -4.96] to (19.68, 196.52, -7.72) mm, rotated rx -180 ry 0 rz 0 deg; joints [26.643, -45.117, 123.589, 27.19, -78.844, -4.968]
  Set speed (500.0 mm/s)
  MoveL 1552 to (19.68, 196.51, 6) mm, rotated rx 180 ry 0 rz 0 deg; joints [26.636, -46.049, 123.777, 27.252, -78.181, -5.314]
  MoveL 1553 to (18.41, 382.85, 6) mm, rotated rx 180 ry 0 rz 0 deg; joints [33.694, -43.253, 115.995, 35.072, -74.852, -9.544]
  Set speed (25.4 mm/s)
  MoveL 1554 to (18.41, 382.85, -4.36) mm, rotated rx 180 ry 0 rz 0 deg; joints [33.7, -42.609, 115.862, 34.999, -75.271, -9.242]
  MoveC 1555 to (18.41, 383.04, -4.81) mm, rotated rx -180 ry 0 rz 0 deg; joints [33.707, -42.578, 115.847, 35.004, -75.286, -9.234] to (18.41, 383.49, -5) mm, rotated rx 180 ry 0 rz 0 deg; joints [33.723, -42.559, 115.824, 35.021, -75.285, -9.24]
  Set speed (50.8 mm/s)
  MoveL 1556 to (18.41, 384.12, -5) mm, rotated rx 180 ry 0 rz 0 deg; joints [33.745, -42.548, 115.794, 35.046, -75.273, -9.257]
  MoveC 1557 to (18.6, 384.57, -5) mm, rotated rx -180 ry 0 rz 0 deg; joints [33.765, -42.545, 115.786, 35.068, -75.272, -9.265] to (19.04, 384.76, -5) mm, rotated rx 180 ry 0 rz 0 deg; joints [33.782, -42.554, 115.809, 35.083, -75.287, -9.261]
  MoveL 1558 to (64.86, 384.76, -5) mm, rotated rx -180 ry 0 rz 0 deg; joints [34.893, -43.761, 118.971, 35.933, -77.053, -8.345]
  MoveL 1559 to (471.26, 384.76, -5) mm, rotated rx -180 ry 0 rz 0 deg; joints [48.234, -51.123, 142.602, 48.223, -90.116, 1.375]
  MoveL 1560 to (471.26, 537.16, -5) mm, rotated rx 180 ry 0 rz 0 deg; joints [53.409, -49.093, 133.877, 53.582, -86.026, -3.923]
  MoveL 1561 to (445.86, 537.16, -5) mm, rotated rx 180 ry 0 rz 0 deg; joints [52.385, -48.73, 132.709, 52.606, -85.463, -4.508]
  MoveC 1562 to (433.16, 524.46, -5) mm, rotated rx -180 ry 0 rz 0 deg; joints [51.489, -48.758, 132.87, 51.702, -85.471, -4.346] to (420.46, 537.16, -5) mm, rotated rx 180 ry 0 rz 0 deg; joints [51.388, -48.347, 131.507, 51.665, -84.872, -5.088]
  MoveL 1563 to (395.06, 537.16, -5) mm, rotated rx -180 ry 0 rz 0 deg; joints [50.418, -47.944, 130.271, 50.757, -84.254, -5.664]
  MoveL 1564 to (318.86, 537.16, -5) mm, rotated rx -180 ry 0 rz 0 deg; joints [47.665, -46.616, 126.36, 48.237, -82.251, -7.36]
  MoveC 1565 to (306.16, 524.46, -5) mm, rotated rx -180 ry 0 rz 0 deg; joints [46.824, -46.616, 126.412, 47.39, -82.175, -7.22] to (293.46, 537.16, -5) mm, rotated rx -180 ry 0 rz 0 deg; joints [46.798, -46.132, 124.99, 47.462, -81.537, -7.915]
  MoveL 1566 to (191.86, 537.16, -5) mm, rotated rx -180 ry 0 rz 0 deg; joints [43.561, -43.992, 119.174, 44.684, -78.463, -10.09]
  MoveC 1567 to (179.16, 524.46, -5) mm, rotated rx 180 ry 0 rz 0 deg; joints [42.777, -43.959, 119.123, 43.899, -78.311, -9.956] to (166.46, 537.16, -5) mm, rotated rx 180 ry 0 rz 0 deg; joints [42.807, -43.405, 117.635, 44.068, -77.644, -10.625]
  MoveL 1568 to (90.26, 537.16, -5) mm, rotated rx 180 ry 0 rz 0 deg; joints [40.668, -41.513, 112.807, 42.4, -75.071, -12.219]
  MoveL 1569 to (64.86, 537.16, -5) mm, rotated rx 180 ry 0 rz 0 deg; joints [39.993, -40.839, 111.125, 41.904, -74.175, -12.749]
  MoveC 1570 to (61.14, 528.18, -5) mm, rotated rx -180 ry 0 rz 0 deg; joints [39.615, -40.931, 111.376, 41.491, -74.209, -12.541] to (52.16, 524.46, -5) mm, rotated rx -180 ry 0 rz 0 deg; joints [39.265, -40.766, 110.975, 41.181, -73.954, -12.611]
  MoveL 1571 to (52.16, 524.46, -5) mm, rotated rx -180 ry 0 rz 0 deg; joints [39.265, -40.766, 110.975, 41.181, -73.954, -12.611]
  MoveC 1572 to (43.18, 528.18, -5) mm, rotated rx 180 ry 0 rz 0 deg; joints [39.152, -40.439, 110.159, 41.159, -73.56, -12.916] to (39.46, 537.16, -5) mm, rotated rx 180 ry 0 rz 0 deg; joints [39.337, -40.141, 109.406, 41.437, -73.261, -13.28]
  MoveL 1573 to (14.06, 537.16, -5) mm, rotated rx 180 ry 0 rz 0 deg; joints [38.699, -39.42, 107.647, 41, -72.328, -13.814]
  MoveL 1574 to (14.06, 384.76, -5) mm, rotated rx 180 ry 0 rz 0 deg; joints [33.665, -42.418, 115.458, 34.996, -75.091, -9.36]
  MoveL 1575 to (19.04, 384.76, -5) mm, rotated rx 180 ry 0 rz 0 deg; joints [33.782, -42.554, 115.809, 35.083, -75.287, -9.261]
  MoveC 1576 to (19.49, 384.57, -5) mm, rotated rx -180 ry 0 rz 0 deg; joints [33.786, -42.569, 115.849, 35.083, -75.307, -9.247] to (19.68, 384.12, -5) mm, rotated rx -180 ry 0 rz 0 deg; joints [33.775, -42.582, 115.883, 35.068, -75.323, -9.232]
  MoveL 1577 to (19.68, 383.49, -5) mm, rotated rx -180 ry 0 rz 0 deg; joints [33.752, -42.593, 115.913, 35.043, -75.335, -9.215]
  MoveC 1578 to (19.68, 383.04, -4.81) mm, rotated rx 180 ry 0 rz 0 deg; joints [33.736, -42.612, 115.936, 35.026, -75.335, -9.209] to (19.68, 382.85, -4.37) mm, rotated rx 180 ry 0 rz 0 deg; joints [33.73, -42.644, 115.951, 35.021, -75.321, -9.217]
  Set speed (500.0 mm/s)
  MoveL 1579 to (19.68, 382.85, 5) mm, rotated rx 180 ry 0 rz 0 deg; joints [33.725, -43.226, 116.072, 35.087, -74.942, -9.49]
  MoveL 1580 to (18.41, 382.85, 5) mm, rotated rx -180 ry 0 rz 0 deg; joints [33.695, -43.191, 115.983, 35.065, -74.893, -9.515]
  Set speed (25.4 mm/s)
  MoveL 1581 to (18.41, 382.85, 1) mm, rotated rx -180 ry 0 rz 0 deg; joints [33.697, -42.943, 115.932, 35.036, -75.055, -9.398]
  MoveL 1582 to (18.41, 382.85, -7.72) mm, rotated rx -180 ry 0 rz 0 deg; joints [33.702, -42.401, 115.817, 34.976, -75.405, -9.145]
  MoveC 1583 to (18.41, 383.04, -8.16) mm, rotated rx -180 ry 0 rz 0 deg; joints [33.708, -42.369, 115.802, 34.981, -75.42, -9.137] to (18.41, 383.49, -8.35) mm, rotated rx 180 ry 0 rz 0 deg; joints [33.724, -42.35, 115.778, 34.998, -75.419, -9.144]
  Set speed (50.8 mm/s)
  MoveL 1584 to (18.41, 384.12, -8.35) mm, rotated rx -180 ry 0 rz 0 deg; joints [33.747, -42.339, 115.749, 35.023, -75.407, -9.16]
  MoveC 1585 to (18.6, 384.57, -8.35) mm, rotated rx -180 ry 0 rz 0 deg; joints [33.767, -42.337, 115.741, 35.045, -75.406, -9.168] to (19.04, 384.76, -8.35) mm, rotated rx -180 ry 0 rz 0 deg; joints [33.784, -42.346, 115.764, 35.06, -75.421, -9.164]
  MoveL 1586 to (64.86, 384.76, -8.35) mm, rotated rx -180 ry 0 rz 0 deg; joints [34.895, -43.545, 118.925, 35.912, -77.191, -8.243]
  MoveL 1587 to (471.26, 384.76, -8.35) mm, rotated rx -180 ry 0 rz 0 deg; joints [48.237, -50.82, 142.543, 48.226, -90.278, 1.557]
  MoveL 1588 to (471.26, 537.16, -8.35) mm, rotated rx -180 ry 0 rz 0 deg; joints [53.411, -48.831, 133.826, 53.573, -86.151, -3.753]
  MoveL 1589 to (445.86, 537.16, -8.35) mm, rotated rx -180 ry 0 rz 0 deg; joints [52.387, -48.472, 132.658, 52.596, -85.589, -4.343]
  MoveC 1590 to (433.16, 524.46, -8.35) mm, rotated rx -180 ry 0 rz 0 deg; joints [51.491, -48.5, 132.819, 51.692, -85.599, -4.183] to (420.46, 537.16, -8.35) mm, rotated rx 180 ry 0 rz 0 deg; joints [51.391, -48.094, 131.457, 51.653, -84.998, -4.929]
  MoveL 1591 to (395.06, 537.16, -8.35) mm, rotated rx -180 ry 0 rz 0 deg; joints [50.421, -47.696, 130.221, 50.744, -84.38, -5.509]
  MoveL 1592 to (318.86, 537.16, -8.35) mm, rotated rx 180 ry 0 rz 0 deg; joints [47.668, -46.38, 126.312, 48.22, -82.376, -7.219]
  MoveC 1593 to (306.16, 524.46, -8.35) mm, rotated rx -180 ry 0 rz 0 deg; joints [46.826, -46.38, 126.364, 47.373, -82.302, -7.081] to (293.46, 537.16, -8.35) mm, rotated rx -180 ry 0 rz 0 deg; joints [46.8, -45.901, 124.942, 47.444, -81.661, -7.778]
  MoveL 1594 to (191.86, 537.16, -8.35) mm, rotated rx 180 ry 0 rz 0 deg; joints [43.563, -43.776, 119.128, 44.662, -78.585, -9.968]
  MoveC 1595 to (179.16, 524.46, -8.35) mm, rotated rx 180 ry 0 rz 0 deg; joints [42.779, -43.743, 119.077, 43.877, -78.434, -9.836] to (166.46, 537.16, -8.35) mm, rotated rx -180 ry 0 rz 0 deg; joints [42.809, -43.192, 117.589, 44.044, -77.764, -10.506]
  MoveL 1596 to (90.26, 537.16, -8.35) mm, rotated rx -180 ry 0 rz 0 deg; joints [40.669, -41.311, 112.763, 42.373, -75.188, -12.109]
  MoveL 1597 to (64.86, 537.16, -8.35) mm, rotated rx 180 ry 0 rz 0 deg; joints [39.995, -40.64, 111.081, 41.876, -74.291, -12.642]
  MoveC 1598 to (61.14, 528.18, -8.35) mm, rotated rx -180 ry 0 rz 0 deg; joints [39.617, -40.732, 111.331, 41.463, -74.325, -12.435] to (52.16, 524.46, -8.35) mm, rotated rx -180 ry 0 rz 0 deg; joints [39.267, -40.568, 110.931, 41.153, -74.071, -12.505]
  MoveL 1599 to (52.16, 524.46, -8.35) mm, rotated rx 180 ry 0 rz 0 deg; joints [39.267, -40.568, 110.931, 41.153, -74.071, -12.505]
  MoveC 1600 to (43.18, 528.18, -8.35) mm, rotated rx -180 ry 0 rz 0 deg; joints [39.154, -40.242, 110.115, 41.132, -73.676, -12.811] to (39.46, 537.16, -8.35) mm, rotated rx 180 ry 0 rz 0 deg; joints [39.339, -39.945, 109.362, 41.409, -73.375, -13.176]
  MoveL 1601 to (14.06, 537.16, -8.35) mm, rotated rx -180 ry 0 rz 0 deg; joints [38.701, -39.228, 107.603, 40.971, -72.441, -13.712]
  MoveL 1602 to (14.06, 384.76, -8.35) mm, rotated rx -180 ry 0 rz 0 deg; joints [33.667, -42.21, 115.413, 34.973, -75.225, -9.264]
  MoveL 1603 to (19.04, 384.76, -8.35) mm, rotated rx -180 ry 0 rz 0 deg; joints [33.784, -42.346, 115.764, 35.06, -75.421, -9.164]
  MoveC 1604 to (19.49, 384.57, -8.35) mm, rotated rx -180 ry 0 rz 0 deg; joints [33.788, -42.361, 115.804, 35.061, -75.442, -9.15] to (19.68, 384.12, -8.35) mm, rotated rx -180 ry 0 rz 0 deg; joints [33.777, -42.374, 115.838, 35.046, -75.457, -9.135]
  MoveL 1605 to (19.68, 383.49, -8.35) mm, rotated rx -180 ry 0 rz 0 deg; joints [33.754, -42.384, 115.868, 35.02, -75.469, -9.118]
  MoveC 1606 to (19.68, 383.04, -8.16) mm, rotated rx -180 ry 0 rz 0 deg; joints [33.738, -42.404, 115.891, 35.003, -75.47, -9.112] to (19.68, 382.85, -7.72) mm, rotated rx -180 ry 0 rz 0 deg; joints [33.731, -42.435, 115.906, 34.999, -75.455, -9.12]
  Set speed (500.0 mm/s)
  MoveL 1607 to (19.68, 382.85, 6) mm, rotated rx -180 ry 0 rz 0 deg; joints [33.724, -43.288, 116.084, 35.094, -74.902, -9.519]
  MoveL 1608 to (-12.15, 384.12, 6) mm, rotated rx 180 ry 0 rz 0 deg; joints [33.033, -42.367, 113.762, 34.613, -73.63, -10.17]
  Set speed (25.4 mm/s)
  MoveL 1609 to (-12.15, 384.12, -4.37) mm, rotated rx -180 ry 0 rz 0 deg; joints [33.038, -41.738, 113.63, 34.536, -74.04, -9.878]
  MoveC 1610 to (-12.34, 384.12, -4.81) mm, rotated rx -180 ry 0 rz 0 deg; joints [33.034, -41.706, 113.611, 34.53, -74.051, -9.869] to (-12.79, 384.12, -5) mm, rotated rx -180 ry 0 rz 0 deg; joints [33.024, -41.682, 113.576, 34.521, -74.04, -9.872]
  Set speed (50.8 mm/s)
  MoveL 1611 to (-13.42, 384.12, -5) mm, rotated rx -180 ry 0 rz 0 deg; joints [33.01, -41.664, 113.531, 34.511, -74.015, -9.885]
  MoveC 1612 to (-13.87, 384.31, -5) mm, rotated rx -180 ry 0 rz 0 deg; joints [33.006, -41.648, 113.49, 34.512, -73.993, -9.899] to (-14.06, 384.76, -5) mm, rotated rx -180 ry 0 rz 0 deg; joints [33.018, -41.635, 113.455, 34.527, -73.978, -9.914]
  MoveL 1613 to (-14.06, 537.16, -5) mm, rotated rx 180 ry 0 rz 0 deg; joints [38.013, -38.595, 105.653, 40.552, -71.273, -14.409]
  MoveL 1614 to (-39.46, 537.16, -5) mm, rotated rx 180 ry 0 rz 0 deg; joints [37.411, -37.823, 103.808, 40.178, -70.3, -14.952]
  MoveC 1615 to (-52.16, 524.46, -5) mm, rotated rx -180 ry 0 rz 0 deg; joints [36.726, -37.715, 103.576, 39.504, -70.025, -14.808] to (-64.86, 537.16, -5) mm, rotated rx -180 ry 0 rz 0 deg; joints [36.825, -37.025, 101.919, 39.834, -69.307, -15.501]
  MoveL 1616 to (-90.26, 537.16, -5) mm, rotated rx -180 ry 0 rz 0 deg; joints [36.254, -36.202, 99.984, 39.521, -68.293, -16.058]
  MoveL 1617 to (-166.46, 537.16, -5) mm, rotated rx -180 ry 0 rz 0 deg; joints [34.631, -33.561, 93.879, 38.774, -65.126, -17.796]
  MoveC 1618 to (-179.16, 524.46, -5) mm, rotated rx 180 ry 0 rz 0 deg; joints [33.995, -33.403, 93.538, 38.16, -64.787, -17.649] to (-191.86, 537.16, -5) mm, rotated rx 180 ry 0 rz 0 deg; joints [34.117, -32.62, 91.734, 38.592, -64.025, -18.405]
  MoveL 1619 to (-293.46, 537.16, -5) mm, rotated rx -180 ry 0 rz 0 deg; joints [32.193, -28.494, 82.491, 38.251, -59.356, -21.072]
  MoveC 1620 to (-306.16, 524.46, -5) mm, rotated rx -180 ry 0 rz 0 deg; joints [31.603, -28.274, 82.02, 37.702, -58.945, -20.932] to (-318.86, 537.16, -5) mm, rotated rx 180 ry 0 rz 0 deg; joints [31.741, -27.358, 79.984, 38.276, -58.113, -21.817]
  MoveL 1621 to (-395.06, 537.16, -5) mm, rotated rx 180 ry 0 rz 0 deg; joints [30.454, -23.633, 71.856, 38.69, -54.155, -24.343]
  MoveL 1622 to (-420.46, 537.16, -5) mm, rotated rx 180 ry 0 rz 0 deg; joints [30.045, -22.262, 68.898, 38.968, -52.745, -25.314]
  MoveC 1623 to (-433.16, 524.46, -5) mm, rotated rx -180 ry 0 rz 0 deg; joints [29.496, -21.951, 68.241, 38.509, -52.239, -25.214] to (-445.86, 537.16, -5) mm, rotated rx -180 ry 0 rz 0 deg; joints [29.646, -20.813, 65.785, 39.334, -51.279, -26.373]
  MoveL 1624 to (-471.26, 537.16, -5) mm, rotated rx 180 ry 0 rz 0 deg; joints [29.257, -19.271, 62.489, 39.806, -49.749, -27.541]
  MoveL 1625 to (-471.26, 384.76, -5) mm, rotated rx 180 ry 0 rz 0 deg; joints [24.973, -23.748, 72.274, 32.244, -52.289, -20.422]
  MoveL 1626 to (-14.06, 384.76, -5) mm, rotated rx 180 ry 0 rz 0 deg; joints [33.018, -41.635, 113.455, 34.527, -73.978, -9.914]
  MoveC 1627 to (-13.61, 384.57, -5) mm, rotated rx 180 ry 0 rz 0 deg; joints [33.021, -41.651, 113.496, 34.526, -73.999, -9.9] to (-13.42, 384.12, -5) mm, rotated rx -180 ry 0 rz 0 deg; joints [33.01, -41.664, 113.531, 34.511, -74.015, -9.885]
  MoveL 1628 to (-13.42, 383.49, -5) mm, rotated rx -180 ry 0 rz 0 deg; joints [32.988, -41.675, 113.56, 34.486, -74.026, -9.868]
  MoveC 1629 to (-13.42, 383.04, -4.81) mm, rotated rx -180 ry 0 rz 0 deg; joints [32.972, -41.694, 113.583, 34.469, -74.027, -9.862] to (-13.42, 382.85, -4.37) mm, rotated rx 180 ry 0 rz 0 deg; joints [32.965, -41.725, 113.598, 34.464, -74.012, -9.869]
  Set speed (500.0 mm/s)
  MoveL 1630 to (-13.42, 382.85, 5) mm, rotated rx -180 ry 0 rz 0 deg; joints [32.96, -42.293, 113.718, 34.533, -73.642, -10.132]
  MoveL 1631 to (-12.15, 384.12, 5) mm, rotated rx 180 ry 0 rz 0 deg; joints [33.034, -42.307, 113.75, 34.605, -73.67, -10.142]
  Set speed (25.4 mm/s)
  MoveL 1632 to (-12.15, 384.12, 1) mm, rotated rx -180 ry 0 rz 0 deg; joints [33.036, -42.064, 113.7, 34.575, -73.829, -10.028]
  MoveL 1633 to (-12.15, 384.12, -7.72) mm, rotated rx -180 ry 0 rz 0 deg; joints [33.04, -41.534, 113.586, 34.512, -74.172, -9.784]
  MoveC 1634 to (-12.34, 384.12, -8.16) mm, rotated rx -180 ry 0 rz 0 deg; joints [33.036, -41.502, 113.566, 34.506, -74.182, -9.775] to (-12.79, 384.12, -8.35) mm, rotated rx -180 ry 0 rz 0 deg; joints [33.026, -41.478, 113.532, 34.498, -74.171, -9.779]
  Set speed (50.8 mm/s)
  MoveL 1635 to (-13.42, 384.12, -8.35) mm, rotated rx 180 ry 0 rz 0 deg; joints [33.012, -41.46, 113.486, 34.487, -74.146, -9.792]
  MoveC 1636 to (-13.87, 384.31, -8.35) mm, rotated rx 180 ry 0 rz 0 deg; joints [33.008, -41.444, 113.445, 34.488, -74.125, -9.806] to (-14.06, 384.76, -8.35) mm, rotated rx 180 ry 0 rz 0 deg; joints [33.019, -41.431, 113.411, 34.503, -74.109, -9.821]
  MoveL 1637 to (-14.06, 537.16, -8.35) mm, rotated rx -180 ry 0 rz 0 deg; joints [38.015, -38.405, 105.61, 40.521, -71.384, -14.31]
  MoveL 1638 to (-39.46, 537.16, -8.35) mm, rotated rx -180 ry 0 rz 0 deg; joints [37.412, -37.636, 103.764, 40.146, -70.409, -14.854]
  MoveC 1639 to (-52.16, 524.46, -8.35) mm, rotated rx 180 ry 0 rz 0 deg; joints [36.728, -37.529, 103.532, 39.473, -70.136, -14.712] to (-64.86, 537.16, -8.35) mm, rotated rx 180 ry 0 rz 0 deg; joints [36.826, -36.842, 101.875, 39.802, -69.415, -15.405]
  MoveL 1640 to (-90.26, 537.16, -8.35) mm, rotated rx 180 ry 0 rz 0 deg; joints [36.255, -36.021, 99.94, 39.488, -68.4, -15.964]
  MoveL 1641 to (-166.46, 537.16, -8.35) mm, rotated rx -180 ry 0 rz 0 deg; joints [34.632, -33.388, 93.835, 38.738, -65.228, -17.707]
  MoveC 1642 to (-179.16, 524.46, -8.35) mm, rotated rx -180 ry 0 rz 0 deg; joints [33.997, -33.23, 93.495, 38.124, -64.889, -17.561] to (-191.86, 537.16, -8.35) mm, rotated rx -180 ry 0 rz 0 deg; joints [34.119, -32.448, 91.69, 38.555, -64.125, -18.318]
  MoveL 1643 to (-293.46, 537.16, -8.35) mm, rotated rx -180 ry 0 rz 0 deg; joints [32.194, -28.331, 82.445, 38.209, -59.449, -20.988]
  MoveC 1644 to (-306.16, 524.46, -8.35) mm, rotated rx -180 ry 0 rz 0 deg; joints [31.604, -28.111, 81.975, 37.661, -59.038, -20.849] to (-318.86, 537.16, -8.35) mm, rotated rx -180 ry 0 rz 0 deg; joints [31.743, -27.197, 79.938, 38.233, -58.204, -21.734]
  MoveL 1645 to (-395.06, 537.16, -8.35) mm, rotated rx -180 ry 0 rz 0 deg; joints [30.455, -23.476, 71.806, 38.644, -54.239, -24.261]
  MoveL 1646 to (-420.46, 537.16, -8.35) mm, rotated rx -180 ry 0 rz 0 deg; joints [30.046, -22.107, 68.847, 38.92, -52.827, -25.232]
  MoveC 1647 to (-433.16, 524.46, -8.35) mm, rotated rx 180 ry 0 rz 0 deg; joints [29.497, -21.796, 68.19, 38.46, -52.321, -25.133] to (-445.86, 537.16, -8.35) mm, rotated rx 180 ry 0 rz 0 deg; joints [29.648, -20.659, 65.732, 39.284, -51.358, -26.291]
  MoveL 1648 to (-471.26, 537.16, -8.35) mm, rotated rx -180 ry 0 rz 0 deg; joints [29.258, -19.117, 62.434, 39.754, -49.826, -27.459]
  MoveL 1649 to (-471.26, 384.76, -8.35) mm, rotated rx 180 ry 0 rz 0 deg; joints [24.974, -23.592, 72.225, 32.201, -52.38, -20.35]
  MoveL 1650 to (-14.06, 384.76, -8.35) mm, rotated rx 180 ry 0 rz 0 deg; joints [33.019, -41.431, 113.411, 34.503, -74.109, -9.821]
  MoveC 1651 to (-13.61, 384.57, -8.35) mm, rotated rx 180 ry 0 rz 0 deg; joints [33.023, -41.447, 113.452, 34.502, -74.131, -9.807] to (-13.42, 384.12, -8.35) mm, rotated rx 180 ry 0 rz 0 deg; joints [33.012, -41.46, 113.486, 34.487, -74.146, -9.792]
  MoveL 1652 to (-13.42, 383.49, -8.35) mm, rotated rx -180 ry 0 rz 0 deg; joints [32.989, -41.471, 113.515, 34.462, -74.157, -9.775]
  MoveC 1653 to (-13.42, 383.04, -8.16) mm, rotated rx 180 ry 0 rz 0 deg; joints [32.974, -41.49, 113.539, 34.445, -74.158, -9.768] to (-13.42, 382.85, -7.72) mm, rotated rx -180 ry 0 rz 0 deg; joints [32.967, -41.521, 113.553, 34.441, -74.144, -9.776]
  Set speed (500.0 mm/s)
  MoveL 1654 to (-13.42, 382.85, 15) mm, rotated rx -180 ry 0 rz 0 deg; joints [32.955, -42.897, 113.837, 34.61, -73.242, -10.418]
  MoveL 1655 to (-13.42, 382.85, 15) mm, rotated rx -180 ry 0 rz 0 deg; joints [32.955, -42.897, 113.837, 34.61, -73.242, -10.418]
